# B&R Automation Studio project NAINV104C00R8L515F00 (part 34)

#### Local.var
```iecst
(*2021-05-18*)
(**)
(*Local Action, State & Status*)
VAR
	eStatus : eFBStatus := Idle;
	udiStatus : UDINT := 0;
END_VAR
(**)
(*Local Alarm*)
VAR
	tyAlmData : tyAlmDat;
	tyInfoData : tyAlmDat;
	tyInfoData1 : tyAlmDat;
	a_tyAlmText : ARRAY[10000..10099] OF tyAlmTxt := [(sAlmText:='New Recipe Not Found In Product Recipe List',sRcyText:='Create New Recipe In Product Setting.'),(sAlmText:='Product Recipe Width Not Match',sRcyText:='Check Product Width And Leader Request Width'),(sAlmText:='New Recipe Not Found In Magazine Recipe List',sRcyText:='Create New Recipe In Magazine Setting.'),(sAlmText:='New Recipe Name Empty',sRcyText:='Request Recipe Name From Leader Is Empty, Check Leader Machine'),96(0)];
END_VAR
(**)
(*Local Output*)
VAR
	bUSAllow : BOOL;
	bDSAllow : BOOL;
	bLeaderSeqCtrlInActive : BOOL;
	bProdAccDataMnl : BOOL;
	bProdUpdtDataMnl : BOOL;
	bMagAccDataMnl : BOOL;
	eTimeAct : eTimeAction;
	bWaitRlsBrd : BOOL;
	tyLeaderInfo : tyLFLeaderInfo;
	tyUpdtProdRcp : tyProdRcpParam;
END_VAR
(**)
(*Local Input*)
VAR
	udiRstErr : UDINT := 0;
	bPrep : BOOL := TRUE;
	bEn : BOOL := TRUE;
	bDis : BOOL := FALSE;
	sIPAddr : STRING[15] := '192.168.0.100';
	sMcNm : STRING[30];
	bAWPrep : BOOL := TRUE;
	bAWDis : BOOL;
	bMnlAccData : BOOL;
	bSectionLeader : BOOL;
	sMagRcpNm : STRING[30];
	diWidthLimit : DINT;
	bWidth2Prep : BOOL;
	bUSWidthChkPrep : BOOL;
	bUSWidthChkEn : BOOL;
	bUSWidthChkSen : BOOL;
	bDSWidthChkPrep : BOOL;
	bDSWidthChkEn : BOOL;
	bDSWidthChkSen : BOOL;
	bProdWidthChk : BOOL;
	bUIProdAccData : BOOL;
	bUIProdUpdtData : BOOL;
	bUIMagAccData : BOOL;
	a_tyProdRcpList : ARRAY[1..c_udiProdRcpMax] OF tyProdRcpParam;
	tyDispProdRcp : tyProdRcpParam;
	tyCurrProdRcp : tyProdRcpParam;
	sCurrMagRcpNm : STRING[30];
	eTimeStat : eTimeAction;
	eTimeStatus : eFBStatus;
	bAccNewRcpCond : BOOL;
	bUpdtNewRcpCond : BOOL;
	bAutoUpdtData : BOOL;
	sInfoMsg : STRING[200];
	bInternalUse : BOOL;
	tyInternalReqProdRcp : tyProdRcpParam;
	bNewBrdEnteredCond : BOOL;
	bOldBrdExitedCond : BOOL;
	bRlsBrd : BOOL;
	tyToLeaderProdRcp : tyProdRcpParam;
	bInternalReqProdRcpDiff : BOOL;
	bUpdtProdRcpDiff : BOOL;
	bRlsBrdProdRcpDiff : BOOL;
	sProgNm : STRING[15] := 'Follower';
	bNtSettingsLoadDone : BOOL := TRUE;
	tOnlineChkDlyTm : TIME;
	bManual : BOOL := FALSE;
	bErr : BOOL := FALSE;
	bWarning : BOOL := FALSE;
	bOps : BOOL := FALSE;
	bStandby : BOOL := FALSE;
	eAWStat : eAWAction;
END_VAR
(**)
(*Local*)
VAR
	bRstErr : BOOL;
	udiRstErrOld : UDINT;
	bInitDone : BOOL;
	bInitialDone : BOOL;
	bAutoAccData : BOOL;
	bProdRcpErr : BOOL;
	bMagRcpErr : BOOL;
	bSetTmErr : BOOL;
	bProdAccDataReq : BOOL;
	sReqProdRcpNm : STRING[254];
	diReqProdRcpWidth : DINT;
	bMagAccDataReq : BOOL;
	sReqMagRcpNm : STRING[30];
	usiProdAccDatStep : USINT;
	usiMagAccDatStep : USINT;
	usiProdUpdtDatStep : USINT;
	tyRlsBrdProdRcpNm : tyProdRcpParam;
	bNewBrdEntered : BOOL;
	bOldBrdExited : BOOL;
	i : INT;
	bSetTm : BOOL;
	fbOnlineChk : fbLFFollowerOnlineChk;
	fbFollower : fbLFFollower;
	tyLeaderToFollowerTag : tyLFLeaderToFollowerTag;
	tyFollowerToLeaderTag : tyLFFollowerToLeaderTag;
	eCurrMachineStat : eMachineStat;
	bLeaderOnline : BOOL;
	bLeaderInfo : BOOL;
	bFollowerInfo : BOOL;
	bProdRcpErrNotExist : BOOL;
	bProdRcpErrWidthMismatch : BOOL;
	bDBAOnWOAlign : BOOL;
	udiModuleNum : UDINT := 3901;
END_VAR
```

#### Act_Alarm.st
```iecst
(** 2019-04-21 **)
ACTION Act_Alarm:

	//Error
	IF EDGEPOS(eStatus = Error) THEN

		tyAlmData.sProgNm		:= p_sProgNm;
		tyAlmData.udiCode		:= udiStatus;
		tyAlmData.eSeverity		:= AlmSeverityError;
		tyAlmData.udiRunTime	:= tyAlmData.udiRunTime + 1;
		tyAlmData.bAlm			:= TRUE;
		tyAlmData.udiModuleNum  := udiModuleNum;
		g_sLFFollowerProgNm		:= p_sProgNm;
		//Get Error Message
		IF tyAlmData.udiCode < 10000 OR tyAlmData.udiCode > 10099 THEN
			tyAlmData.sAlmMsg	:= 'Unknown';
			tyAlmData.sRcyMsg	:= 'Unknown';
		ELSE
			tyAlmData.sAlmMsg	:= a_tyAlmText[tyAlmData.udiCode].sAlmText;
			tyAlmData.sRcyMsg	:= a_tyAlmText[tyAlmData.udiCode].sRcyText;
		END_IF

	ELSIF bRstErr AND (tyAlmData.udiCode <> 0) THEN

		tyAlmData.udiCode	:= 0;
		tyAlmData.eSeverity	:= AlmSeverityNA;
		tyAlmData.sAlmMsg	:= '';
		tyAlmData.sRcyMsg	:= '';
		tyAlmData.bAlm			:= FALSE;
	END_IF

END_ACTION
```

#### Act_Background.st
```iecst
(** 2021-05-18 **)
ACTION Act_Background:

	IF p_bInternalUse = TRUE THEN
		tyLeaderToFollowerTag.sReqProdRcpNm		:= p_tyInternalReqProdRcp.sRcpNm;
		IF p_bWidth2Prep THEN
			tyLeaderToFollowerTag.diReqProdRcpWidth	:= p_tyInternalReqProdRcp.diWidthInUM2;
		ELSE
			tyLeaderToFollowerTag.diReqProdRcpWidth	:= p_tyInternalReqProdRcp.diWidthInUM;
		END_IF
		tyLeaderToFollowerTag.sReqMagRcpNm		:= '';
		tyLeaderToFollowerTag.bMnlAccData		:= FALSE;
		tyLeaderToFollowerTag.bBypassMnlAccData	:= FALSE;
		tyLeaderToFollowerTag.bBlkDS			:= FALSE;
		tyLeaderToFollowerTag.bBlkUS			:= FALSE;
		tyLeaderToFollowerTag.bBypassWidthChk	:= TRUE;
		tyLeaderToFollowerTag.bSetTm			:= FALSE;
		tyLeaderToFollowerTag.dtTm				:= 0;
		tyLeaderToFollowerTag.uiTmZone			:= 0;
		tyLeaderToFollowerTag.usiRunTm			:= 0;
		tyLeaderToFollowerTag.bProdNameUSWarn	:= FALSE;
		tyLeaderToFollowerTag.bProdNameDSWarn	:= FALSE;
		tyLeaderToFollowerTag.bProdWidthUSWarn	:= FALSE;
		tyLeaderToFollowerTag.bProdWidthDSWarn	:= FALSE;
		tyLeaderToFollowerTag.bLeaderSeqCtrlInActive	:= FALSE;
	END_IF

	Act_Background_UpdtData;

	//FB
	fbFollower.tyLeaderToFollowerTag	:= tyLeaderToFollowerTag;
	fbFollower.sMcNm					:= p_sMcNm;
	fbFollower.sIPAddr					:= p_sIPAddr;
	fbFollower.bSectionLeader			:= p_bSectionLeader;
	fbFollower.sCurrProdRcpNm			:= p_tyCurrProdRcp.sRcpNm;
	fbFollower.diCurrProdWidthUS		:= p_tyCurrProdRcp.diWidthInUM;
	fbFollower.diCurrProdWidthDS		:= p_tyCurrProdRcp.diWidthInUM2;
	fbFollower.sCurrMagRcpNm			:= p_sCurrMagRcpNm;
	fbFollower.sUpdtLeaderProdRcpNm		:= p_tyToLeaderProdRcp.sRcpNm;
	fbFollower.diUpdtLeaderProdWidthUS	:= p_tyToLeaderProdRcp.diWidthInUM;
	fbFollower.diUpdtLeaderProdWidthDS	:= p_tyToLeaderProdRcp.diWidthInUM2;
	fbFollower.sUpdtLeaderMagRcpNm		:= p_sMagRcpNm;
	fbFollower.bMnlAccDat				:= p_bMnlAccData;
	fbFollower.bAWEn					:= (p_bAWPrep = TRUE) AND (p_bAWDis = FALSE);
	fbFollower.bUSWidthChkEn			:= p_bUSWidthChkPrep AND p_bUSWidthChkEn;
	fbFollower.bUSWidthChkSen			:= p_bUSWidthChkSen;
	fbFollower.bDSWidthChkEn			:= p_bDSWidthChkPrep AND p_bDSWidthChkEn;
	fbFollower.bDSWidthChkSen			:= p_bDSWidthChkSen;
	fbFollower.bProdWidthChk			:= p_bProdWidthChk;
	fbFollower.bProdRcpErr				:= bProdRcpErr;
	fbFollower.bMagRcpErr				:= bMagRcpErr;
	fbFollower.bSetTmErr				:= bSetTmErr;
	fbFollower.eCurrMachineStat			:= eCurrMachineStat;
	fbFollower.bProdChgOverActive		:= (p_eAWStat = AWActGoWidthOff);
	fbFollower.bDBAOnWOAlign			:= p_bDBAOnWOAlign;

	fbFollower(bEn := TRUE);

	tyFollowerToLeaderTag	:= fbFollower.tyFollowerToLeaderTag;
	bProdAccDataReq			:= fbFollower.bProdAccDataReq OR (p_bInternalReqProdRcpDiff = TRUE) ;
	bMagAccDataReq			:= fbFollower.bMagAccDataReq;
	bAutoAccData			:= fbFollower.bAutoAccData;

	IF p_bInternalUse THEN
		bLeaderOnline			:= TRUE;
	ELSE
		bLeaderOnline			:= tyLeaderInfo.bOnline;
	END_IF

	IF bLeaderOnline=FALSE THEN
		bUSAllow				:= TRUE;
		bDSAllow				:= TRUE;
		bLeaderSeqCtrlInActive	:= FALSE;
	ELSE
		bUSAllow				:= fbFollower.bUSAllow AND (p_bInternalReqProdRcpDiff = FALSE);
		bDSAllow				:= fbFollower.bDSAllow;
		bLeaderSeqCtrlInActive	:= tyLeaderToFollowerTag.bLeaderSeqCtrlInActive;
	END_IF

	fbOnlineChk.tyLeaderToFollowerTag	:= tyLeaderToFollowerTag;
	fbOnlineChk(bEn := TRUE);

	Act_Background_AccData;
	Act_Background_ChkRlsBrd;

	//Set Time
	IF EDGEPOS(tyLeaderToFollowerTag.bSetTm) THEN
		bSetTm	:= TRUE;
	END_IF

	IF bSetTm = TRUE THEN
		eTimeAct	:= TimeActSetTime;

		IF (p_eTimeStat = TimeActSetTime) AND (p_eTimeStatus = Done) THEN
			eTimeAct		:= TimeActIdle;
			bSetTm			:= FALSE;
		ELSIF p_eTimeStatus = Error THEN
			eTimeAct		:= TimeActIdle;
			bSetTm			:= FALSE;
		END_IF
	END_IF

	bSetTmErr	:= p_eTimeStatus = Error;

	IF (eStatus = Error) AND bRstErr THEN
		eStatus		:= Idle;
		udiStatus	:= 0;
		bProdRcpErr	:= FALSE;
		bProdRcpErrNotExist	:= FALSE;
		bProdRcpErrWidthMismatch:= FALSE;
		bMagRcpErr	:= FALSE;
	END_IF

END_ACTION
```

#### Act_Background_AccData.st
```iecst
(** 2023-02-22 **)
ACTION Act_Background_AccData:
	//Product Accept Data Request
	CASE usiProdAccDatStep OF
		0:
			//Check Error & Request Accept Data
			// If Product Name/Width Error, Check In Background To Update Data
			IF ((eStatus <> Error) AND (bProdAccDataReq = TRUE)) OR bProdRcpErr THEN
				sReqProdRcpNm		:= tyLeaderToFollowerTag.sReqProdRcpNm;
				diReqProdRcpWidth	:= tyLeaderToFollowerTag.diReqProdRcpWidth;
				usiProdAccDatStep	:= 1;
			END_IF

			IF bLeaderOnline=FALSE THEN
				tyInfoData.sProgNm		:= '';
				tyInfoData.udiCode		:= 0;
				tyInfoData.eSeverity	:= AlmSeverityNA;
				tyInfoData.sAlmMsg		:= '';

				bProdRcpErr 			:= FALSE;
				bProdRcpErrNotExist		:= FALSE;
				bProdRcpErrWidthMismatch:= FALSE;
			END_IF

		1:
			IF p_bInternalUse THEN
				usiProdAccDatStep	:= 2;
			ELSE
				//Check In List Of Recipe
				FOR i := 1 TO 2000 DO
					IF sReqProdRcpNm = '' THEN
						EXIT;
					ELSIF sReqProdRcpNm = pa_tyProdRcpList[i].sRcpNm  THEN
						EXIT;
					END_IF
				END_FOR

				IF sReqProdRcpNm = pa_tyProdRcpList[i].sRcpNm AND diReqProdRcpWidth <> pa_tyProdRcpList[i].diWidthInUM THEN
					//Width Mismatch
					bProdRcpErr := TRUE;
					bProdRcpErrWidthMismatch:= TRUE;
					bProdRcpErrNotExist		:= FALSE;
					usiProdAccDatStep	:= 0;
				ELSIF i > 2000 THEN
					//Recipe Not Exist
					bProdRcpErr := TRUE;
					bProdRcpErrNotExist	:= TRUE;
					bProdRcpErrWidthMismatch:= FALSE;
					usiProdAccDatStep	:= 0;
				ELSE
					bProdRcpErr := FALSE;
					bProdRcpErrNotExist	:= FALSE;
					bProdRcpErrWidthMismatch:= FALSE;
					usiProdAccDatStep	:= 2;
				END_IF

				//Info Message
				IF bLeaderOnline=FALSE THEN
					tyInfoData.sProgNm		:= '';
					tyInfoData.udiCode		:= 0;
					tyInfoData.eSeverity	:= AlmSeverityNA;
					tyInfoData.sAlmMsg		:= '';

					bProdRcpErr 			:= FALSE;
					bProdRcpErrNotExist		:= FALSE;
					bProdRcpErrWidthMismatch:= FALSE;
				ELSE

					IF p_bInternalUse = FALSE THEN
						IF bLeaderInfo OR bFollowerInfo THEN
							tyInfoData.sProgNm		:= p_sProgNm;
							tyInfoData.udiCode		:= 10000;
							tyInfoData.eSeverity	:= AlmSeverityInfo;
							tyInfoData.sAlmMsg		:= p_sInfoMsg;
						ELSE
							tyInfoData.sProgNm		:= '';
							tyInfoData.udiCode		:= 0;
							tyInfoData.eSeverity	:= AlmSeverityNA;
							tyInfoData.sAlmMsg		:= '';
						END_IF
					ELSE
						IF p_sInfoMsg <> '' THEN
							tyInfoData.sProgNm		:= p_sProgNm;
							tyInfoData.udiCode		:= 10000;
							tyInfoData.eSeverity	:= AlmSeverityInfo;
							tyInfoData.sAlmMsg		:= p_sInfoMsg;
						ELSE
							tyInfoData.sProgNm		:= '';
							tyInfoData.udiCode		:= 0;
							tyInfoData.eSeverity	:= AlmSeverityNA;
							tyInfoData.sAlmMsg		:= '';
						END_IF

					END_IF
				END_IF
			END_IF
		2:
			//Manual Accept Data Check
			IF bProdAccDataReq = TRUE THEN
				IF bAutoAccData = FALSE THEN
					bProdAccDataMnl	:= TRUE;

					//Info Message
					IF bLeaderOnline=FALSE THEN
						tyInfoData.sProgNm		:= '';
						tyInfoData.udiCode		:= 0;
						tyInfoData.eSeverity	:= AlmSeverityNA;
						tyInfoData.sAlmMsg		:= '';
					ELSE
						IF p_sInfoMsg <> '' THEN
							tyInfoData.sProgNm		:= p_sProgNm;
							tyInfoData.udiCode		:= 10000;
							tyInfoData.eSeverity	:= AlmSeverityInfo;
							tyInfoData.sAlmMsg		:= p_sInfoMsg;
						ELSE
							tyInfoData.sProgNm		:= '';
							tyInfoData.udiCode		:= 0;
							tyInfoData.eSeverity	:= AlmSeverityNA;
							tyInfoData.sAlmMsg		:= '';
						END_IF
					END_IF

					IF p_bUIProdAccData = TRUE THEN
						p_bUIProdAccData 	:= FALSE; //2023_07_26_Debug for Manual Accept Data automatically accept after product change many times
						bProdAccDataMnl		:= FALSE;
						usiProdAccDatStep	:= 3;
					END_IF
				ELSE
					bProdAccDataMnl		:= FALSE;
					p_bUIProdAccData	:= FALSE; //2023_07_26_Debug for Manual Accept Data automatically accept after product change many times
					usiProdAccDatStep	:= 3;
				END_IF
			ELSE
				bProdAccDataMnl		:= FALSE;
				usiProdAccDatStep	:= 6;
			END_IF

		3:
			//Accept New Recipe Condition
			IF bProdAccDataReq = TRUE THEN
				IF p_bAccNewRcpCond = TRUE THEN

					usiProdAccDatStep	:= 4;
				ELSE
					//Info Message
					IF bLeaderOnline=FALSE THEN
						tyInfoData.sProgNm		:= '';
						tyInfoData.udiCode		:= 0;
						tyInfoData.eSeverity	:= AlmSeverityNA;
						tyInfoData.sAlmMsg		:= '';
					ELSE
						IF p_sInfoMsg <> '' THEN
							tyInfoData.sProgNm		:= p_sProgNm;
							tyInfoData.udiCode		:= 10000;
							tyInfoData.eSeverity	:= AlmSeverityInfo;
							tyInfoData.sAlmMsg		:= p_sInfoMsg;
						ELSE
							tyInfoData.sProgNm		:= '';
							tyInfoData.udiCode		:= 0;
							tyInfoData.eSeverity	:= AlmSeverityNA;
							tyInfoData.sAlmMsg		:= '';
						END_IF
					END_IF
				END_IF
			ELSE
				usiProdAccDatStep	:= 6;
			END_IF

		4:
			//Accept New Recipe Name
			IF p_bInternalUse = TRUE THEN

				p_tyCurrProdRcp	:= p_tyInternalReqProdRcp;
				usiProdAccDatStep := 6;
			ELSE

				FOR i := 1 TO 2000 DO
					IF sReqProdRcpNm = '' THEN
						EXIT;
					ELSIF sReqProdRcpNm = pa_tyProdRcpList[i].sRcpNm THEN
						p_tyCurrProdRcp	:= pa_tyProdRcpList[i];

						EXIT;
					END_IF
				END_FOR

				IF i > 2000 THEN
					//Recipe Not Exist
					bProdRcpErr := TRUE;
					bProdRcpErrNotExist	:= TRUE;
				END_IF
				usiProdAccDatStep	:= 5;
			END_IF

		5:
			(* Add *)
			p_tyProdRcpCurrRcpWr 	:= p_tyCurrProdRcp;
			p_eLinkUIProdRcpAct 	:= ProdRcpActWriteCurrRcpParam;

			IF p_eProdRcpStat = ProdRcpActWriteCurrRcpParam AND p_eProdRcpStatus = Done THEN
				p_eLinkUIProdRcpAct := ProdRcpActIdle;
				usiProdAccDatStep := 6;
			END_IF

		6:
			//Clear Info Message
			tyInfoData.sProgNm		:= '';
			tyInfoData.udiCode		:= 0;
			tyInfoData.eSeverity	:= AlmSeverityNA;
			tyInfoData.sAlmMsg		:= '';

			usiProdAccDatStep	:= 0;

	END_CASE

END_ACTION
```

#### Act_Background_UpdtData.st
```iecst
(** 2019-07-04 **)
ACTION Act_Background_UpdtData:

	//Update To Leader Recipe
	CASE usiProdUpdtDatStep OF
		0:
			//Update New Recipe Condition
			IF tyUpdtProdRcp.sRcpNm <> '' THEN
				IF (p_tyCurrProdRcp.sRcpNm <> tyUpdtProdRcp.sRcpNm) OR (p_bUpdtProdRcpDiff = TRUE) THEN
					IF p_bUpdtNewRcpCond = TRUE THEN
						usiProdUpdtDatStep	:= 1;
					END_IF
				END_IF
			ELSE
				tyUpdtProdRcp	:= p_tyCurrProdRcp;
			END_IF

		1:
			//Manual Update Data Check
			IF p_bAutoUpdtData = FALSE THEN
				bProdUpdtDataMnl	:= TRUE;

				IF p_bUIProdUpdtData = TRUE THEN
					bProdUpdtDataMnl	:= FALSE;
					usiProdUpdtDatStep	:= 2;
				END_IF
			ELSE
				bProdUpdtDataMnl	:= FALSE;
				usiProdUpdtDatStep	:= 2;
			END_IF

		2:
			//Update New Recipe
			tyUpdtProdRcp	:= p_tyCurrProdRcp;

			usiProdUpdtDatStep	:= 0;

	END_CASE

END_ACTION
```

#### Act_InitGlobal.st
```iecst
(** 2020-08-06 **)
ACTION Act_InitGlobal:

	(* Always Change If Project Change *)

	//Pass Data To Link
	p_bLinkStartupRun ACCESS p_StartupRun;
	p_eLinkMcParamUSCommMod ACCESS p_McParamUSCommMod;

	p_bLinkOpsRun ACCESS p_OpsRun;
	p_bLinkConvHvBrd ACCESS p_OpsInvertHvBrd;
	p_bLinkUSWidthChkSen ACCESS p_DIUSWidthChkSen;
	p_bLinkUSWidthChkSen1 ACCESS p_DIUSWidthChkSen1;
	p_bLinkDIInvertHomeSen ACCESS p_DIInvertHomeSen;
	p_bLinkDIInvertRemoteSen ACCESS p_DIInvertRemoteSen;

	//Pass Data To Internal Use
	p_udiRstErr ACCESS p_RstErrReset;
	p_bPrep ACCESS p_NtParamLFPrep;
	p_bEn ACCESS p_McParamLFEn;
	p_sIPAddr ACCESS p_HWInfoIPAddr;
	p_sMcNm ACCESS p_McParamMcNm;
	p_bAWPrep ACCESS p_NtParamAWPrep;
	p_bAWDis ACCESS p_McParamAWDis;
	p_bMnlAccData ACCESS p_McParamMnlAccDat;
	p_bSectionLeader ACCESS p_McParamSectionLeader;
	p_diWidthLimit ACCESS p_NtParamLFWidthLimit;
	p_bUSWidthChkPrep ACCESS p_NtParamUSWidthChkPrep;
	p_bUSWidthChkEn ACCESS p_McParamUSWidthChkEn;
//	p_bUSWidthChkSen ACCESS p_DIUSWidthChkSen;
	p_bDSWidthChkPrep ACCESS p_NtParamDSWidthChkPrep;
	p_bDSWidthChkEn ACCESS p_McParamDSWidthChkEn;
	p_bDSWidthChkSen ACCESS p_DIDSWidthChkSen;
	p_bProdWidthChk ACCESS p_NtParamLFProdWidthChk;
	p_bUIProdAccData ACCESS p_UIProdAccData;
	p_bUIProdUpdtData ACCESS p_UIProdAccData;
	pa_tyProdRcpList ACCESS p_ProdRcpCurrList;
	p_tyCurrProdRcp ACCESS p_ProdRcpCurrRcp0;
	p_tyDispProdRcp ACCESS p_ProdRcpCurrRcp1;
	p_eTimeStat ACCESS p_TimeStat;
	p_eTimeStatus ACCESS p_TimeStatus;
	p_tyToLeaderProdRcp ACCESS p_Follower1UpdtProdRcp;	//Assign With Conveyor Last Zone (To Leader Completion Update)
	p_sProgNm ACCESS p_NtParamLFFollowerProgNm;
	p_bNtSettingsLoadDone ACCESS p_StartupNtSettingsLoadDone;

	p_tOnlineChkDlyTm ACCESS p_NtParamLFFllowerOnlineChkDlyTm;
	p_bManual ACCESS p_UIUIMnlMod;
	p_bErr ACCESS p_AlarmErr;
	p_bOps ACCESS p_OpsStatusRun;
	p_bStandby ACCESS p_OpsStatusStop;
	p_bWarning ACCESS p_AlarmWarning;
	p_eAWStat ACCESS p_AWOpenStat;
	p_bWidth2Prep ACCESS p_NtParamLFWidth2Prep;
	p_bDBAOnWOAlign ACCESS p_McParamDBAOnWOAlign;

	// Add for remain last Loaded product after power cycle
	p_eProdRcpStat ACCESS p_ProdRcpStat;
	p_eProdRcpStatus ACCESS p_ProdRcpStatus;
	p_eLinkUIProdRcpAct ACCESS p_UIProdRcpAct;
	p_tyProdRcpCurrRcpWr ACCESS p_UIProdRcpCurrRcpWr;

	(* Always Change If Project Change *)

END_ACTION
```

#### Act_Initial.st
```iecst
(** 2020-08-06 **)
ACTION Act_Initial:

	//Initial
	fbFollower.diWidthLimit	:= p_diWidthLimit;
	fbFollower(bEn := FALSE);

	fbOnlineChk.p_tyLeaderInfo		:= ADR(tyLeaderInfo);
	fbOnlineChk.tDlyTm				:= p_tOnlineChkDlyTm;
	fbOnlineChk(bEn := FALSE);

END_ACTION
```

#### Act_InitLocal.st
```iecst
(** 2021-05-18 **)
ACTION Act_InitLocal:

	//Input Reference Link To Local Variable
	p_udiRstErr ACCESS ADR(udiRstErr);
	p_bPrep ACCESS ADR(bPrep);
	p_bEn ACCESS ADR(bEn);
	p_bDis ACCESS ADR(bDis);
	p_sIPAddr ACCESS ADR(sIPAddr);
	p_sMcNm ACCESS ADR(sMcNm);
	p_bAWPrep ACCESS ADR(bAWPrep);
	p_bAWDis ACCESS ADR(bAWDis);
	p_bMnlAccData ACCESS ADR(bMnlAccData);
	p_bSectionLeader ACCESS ADR(bSectionLeader);
	p_sMagRcpNm ACCESS ADR(sMagRcpNm);
	p_diWidthLimit ACCESS ADR(diWidthLimit);
	p_bUSWidthChkPrep ACCESS ADR(bUSWidthChkPrep);
	p_bUSWidthChkEn ACCESS ADR(bUSWidthChkEn);
	p_bUSWidthChkSen ACCESS ADR(bUSWidthChkSen);
	p_bDSWidthChkPrep ACCESS ADR(bDSWidthChkPrep);
	p_bDSWidthChkEn ACCESS ADR(bDSWidthChkEn);
	p_bDSWidthChkSen ACCESS ADR(bDSWidthChkSen);
	p_bProdWidthChk ACCESS ADR(bProdWidthChk);
	p_bUIProdAccData ACCESS ADR(bUIProdAccData);
	p_bUIProdUpdtData ACCESS ADR(bUIProdUpdtData);
	p_bUIMagAccData ACCESS ADR(bUIMagAccData);
	pa_tyProdRcpList ACCESS ADR(a_tyProdRcpList);
	p_tyCurrProdRcp ACCESS ADR(tyCurrProdRcp);
	p_tyDispProdRcp ACCESS ADR(tyDispProdRcp);
	p_sCurrMagRcpNm ACCESS ADR(sCurrMagRcpNm);
	p_eTimeStat ACCESS ADR(eTimeStat);
	p_eTimeStatus ACCESS ADR(eTimeStatus);
	p_bAccNewRcpCond ACCESS ADR(bAccNewRcpCond);
	p_bUpdtNewRcpCond ACCESS ADR(bUpdtNewRcpCond);
	p_bAutoUpdtData ACCESS ADR(bAutoUpdtData);
	p_sInfoMsg ACCESS ADR(sInfoMsg);
	p_bInternalUse ACCESS ADR(bInternalUse);
	p_tyInternalReqProdRcp ACCESS ADR(tyInternalReqProdRcp);
	p_bNewBrdEnteredCond ACCESS ADR(bNewBrdEnteredCond);
	p_bOldBrdExitedCond ACCESS ADR(bOldBrdExitedCond);
	p_bRlsBrd ACCESS ADR(bRlsBrd);
	p_tyToLeaderProdRcp ACCESS ADR(tyToLeaderProdRcp);
	p_bInternalReqProdRcpDiff ACCESS ADR(bInternalReqProdRcpDiff);
	p_bUpdtProdRcpDiff ACCESS ADR(bUpdtProdRcpDiff);
	p_bRlsBrdProdRcpDiff ACCESS ADR(bRlsBrdProdRcpDiff);
	p_sProgNm ACCESS ADR(sProgNm);
	p_bNtSettingsLoadDone ACCESS ADR(bNtSettingsLoadDone);
	p_tOnlineChkDlyTm ACCESS ADR(tOnlineChkDlyTm);
	p_bManual ACCESS ADR(bManual);
	p_bErr ACCESS ADR(bErr);
	p_bWarning ACCESS ADR(bWarning);
	p_bOps ACCESS ADR(bOps);
	p_bStandby ACCESS ADR(bStandby);
	p_eAWStat ACCESS ADR(eAWStat);
	p_bWidth2Prep ACCESS ADR(bWidth2Prep);
	p_bDBAOnWOAlign ACCESS ADR(bDBAOnWOAlign);
END_ACTION
```

#### Act_Link.st
```iecst
(** 2021-05-18 **)
ACTION Act_Link:

	bFollowerInfo	:= tyFollowerToLeaderTag.bProdWidthErr OR bProdRcpErrNotExist OR bProdRcpErrWidthMismatch;

	bLeaderInfo		:= (tyLeaderToFollowerTag.bProdWidthUSWarn OR tyLeaderToFollowerTag.bProdWidthDSWarn
						OR ((tyLeaderToFollowerTag.bProdNameUSWarn OR tyLeaderToFollowerTag.bProdNameDSWarn)
						AND (p_bAWPrep = TRUE) AND (p_bAWDis = FALSE) AND (p_eAWStat<>AWActGoWidthOff)));

	//Info Message
	IF bFollowerInfo THEN
		IF tyFollowerToLeaderTag.bProdWidthErr = TRUE OR bProdRcpErrWidthMismatch THEN

			p_sInfoMsg		:= 'Product Recipe Width Does Not Match';
			p_sInfoMsg		:= CONCAT(p_sInfoMsg , '$r$n');
			p_sInfoMsg		:= CONCAT(p_sInfoMsg , 'Check Product Width And');
			p_sInfoMsg		:= CONCAT(p_sInfoMsg , '$r$n');
			p_sInfoMsg		:= CONCAT(p_sInfoMsg , 'Leader Request Width');

		ELSIF bProdRcpErrNotExist THEN

			p_sInfoMsg		:= 'New Product Not Found';
			p_sInfoMsg		:= CONCAT(p_sInfoMsg , '$r$n');
			p_sInfoMsg		:= CONCAT(p_sInfoMsg , 'In Product Recipe List');
			p_sInfoMsg		:= CONCAT(p_sInfoMsg , '$r$n');
			p_sInfoMsg		:= CONCAT(p_sInfoMsg , 'Create New Product');
			p_sInfoMsg		:= CONCAT(p_sInfoMsg , '$r$n');
			p_sInfoMsg		:= CONCAT(p_sInfoMsg , 'In Product Setting');
		END_IF
	ELSE

		IF (tyLeaderToFollowerTag.sReqProdRcpNm<>p_tyCurrProdRcp.sRcpNm) AND (tyLeaderToFollowerTag.sReqProdRcpNm<>'')
			AND bLeaderInfo=FALSE THEN

			p_sInfoMsg		:= 'Leader Request New Recipe';
			p_sInfoMsg		:= CONCAT(p_sInfoMsg , '$r$n');
			p_sInfoMsg		:= CONCAT(p_sInfoMsg , 'Old Recipe Name : ');
			p_sInfoMsg		:= CONCAT(p_sInfoMsg , p_tyDispProdRcp.sRcpNm);
			p_sInfoMsg		:= CONCAT(p_sInfoMsg , '$r$n');
			p_sInfoMsg		:= CONCAT(p_sInfoMsg , 'Old Recipe Width : ');
			sWidthInUMTemp	:= DINT_TO_STRING(p_tyDispProdRcp.diWidthInUM / 1000);
			p_sInfoMsg		:= CONCAT(p_sInfoMsg , sWidthInUMTemp);
			p_sInfoMsg		:= CONCAT(p_sInfoMsg , '$r$n');
			p_sInfoMsg		:= CONCAT(p_sInfoMsg , 'New Recipe Name : ');
			p_sInfoMsg		:= CONCAT(p_sInfoMsg , tyLeaderToFollowerTag.sReqProdRcpNm);
			p_sInfoMsg		:= CONCAT(p_sInfoMsg , '$r$n');
			p_sInfoMsg		:= CONCAT(p_sInfoMsg , 'New Recipe Width : ');
			sWidthInUMTemp	:= DINT_TO_STRING(tyLeaderToFollowerTag.diReqProdRcpWidth / 1000);
			p_sInfoMsg		:= CONCAT(p_sInfoMsg , sWidthInUMTemp);

		ELSIF tyLeaderToFollowerTag.bProdNameUSWarn THEN
			p_sInfoMsg		:= 'US Machine Request New Recipe';
			p_sInfoMsg		:= CONCAT(p_sInfoMsg , '$r$n');
			p_sInfoMsg		:= CONCAT(p_sInfoMsg , 'Old Recipe Name : ');
			p_sInfoMsg		:= CONCAT(p_sInfoMsg , p_tyDispProdRcp.sRcpNm);
			p_sInfoMsg		:= CONCAT(p_sInfoMsg , '$r$n');
			p_sInfoMsg		:= CONCAT(p_sInfoMsg , 'Old Recipe Width : ');
			sWidthInUMTemp	:= DINT_TO_STRING(p_tyDispProdRcp.diWidthInUM / 1000);
			p_sInfoMsg		:= CONCAT(p_sInfoMsg , sWidthInUMTemp);
			p_sInfoMsg		:= CONCAT(p_sInfoMsg , '$r$n');
			p_sInfoMsg		:= CONCAT(p_sInfoMsg , 'New Recipe Name : ');
			p_sInfoMsg		:= CONCAT(p_sInfoMsg , tyLeaderToFollowerTag.sReqProdRcpNm);
			p_sInfoMsg		:= CONCAT(p_sInfoMsg , '$r$n');
			p_sInfoMsg		:= CONCAT(p_sInfoMsg , 'New Recipe Width : ');
			sWidthInUMTemp	:= DINT_TO_STRING(tyLeaderToFollowerTag.diReqProdRcpWidth / 1000);
			p_sInfoMsg		:= CONCAT(p_sInfoMsg , sWidthInUMTemp);

		ELSIF tyLeaderToFollowerTag.bProdNameDSWarn THEN
			p_sInfoMsg		:= 'Different Recipe';
			p_sInfoMsg		:= CONCAT(p_sInfoMsg , '$r$n');
			p_sInfoMsg		:= CONCAT(p_sInfoMsg , 'From DS Machine');
			p_sInfoMsg		:= CONCAT(p_sInfoMsg , '$r$n');
			p_sInfoMsg		:= CONCAT(p_sInfoMsg , 'Current Recipe Name : ');
			p_sInfoMsg		:= CONCAT(p_sInfoMsg , p_tyCurrProdRcp.sRcpNm);
			p_sInfoMsg		:= CONCAT(p_sInfoMsg , '$r$n');
			p_sInfoMsg		:= CONCAT(p_sInfoMsg , 'Current Recipe Width : ');
			sWidthInUMTemp	:= DINT_TO_STRING(p_tyCurrProdRcp.diWidthInUM2 / 1000);
			p_sInfoMsg		:= CONCAT(p_sInfoMsg , sWidthInUMTemp);

		ELSIF tyLeaderToFollowerTag.bProdWidthUSWarn THEN
			p_sInfoMsg		:= 'Product Recipe Width Does Not Match';
			p_sInfoMsg		:= CONCAT(p_sInfoMsg , '$r$n');
			p_sInfoMsg		:= CONCAT(p_sInfoMsg , 'Check Product Width And');
			p_sInfoMsg		:= CONCAT(p_sInfoMsg , '$r$n');
			p_sInfoMsg		:= CONCAT(p_sInfoMsg , 'Leader Request Width');

		ELSIF tyLeaderToFollowerTag.bProdWidthDSWarn THEN
			p_sInfoMsg		:= 'Same Recipe : ';
			p_sInfoMsg		:= CONCAT(p_sInfoMsg , p_tyDispProdRcp.sRcpNm);
			p_sInfoMsg		:= CONCAT(p_sInfoMsg , '$r$n');
			p_sInfoMsg		:= CONCAT(p_sInfoMsg , 'But Different Width');
			p_sInfoMsg		:= CONCAT(p_sInfoMsg , '$r$n');
			p_sInfoMsg		:= CONCAT(p_sInfoMsg , 'With DS Machine');
			p_sInfoMsg		:= CONCAT(p_sInfoMsg , '$r$n');
			p_sInfoMsg		:= CONCAT(p_sInfoMsg , 'Machine Outgoing Width : ');
			sWidthInUMTemp	:= DINT_TO_STRING(p_tyDispProdRcp.diWidthInUM2 / 1000);
			p_sInfoMsg		:= CONCAT(p_sInfoMsg , sWidthInUMTemp);

		END_IF
	END_IF

	//Accept New Recipe Condition (Before Loaded New Recipe)
	p_bAccNewRcpCond	:= p_bLinkOpsRun = TRUE AND p_bLinkConvHvBrd = FALSE;

	//Update New Recipe Condition (After Loaded New Recipe)
	p_bUpdtNewRcpCond	:= TRUE;

	//Recipe Different
	//p_bInternalReqProdRcpDiff	:= memcmp(ADR(p_tyCurrProdRcp) , ADR(p_tyInternalReqProdRcp) , SIZEOF(p_tyCurrProdRcp)) <> 0;
	//p_bUpdtProdRcpDiff		:= memcmp(ADR(p_tyCurrProdRcp) , ADR(tyUpdtProdRcp) , SIZEOF(p_tyCurrProdRcp)) <> 0;
	//p_bRlsBrdProdRcpDiff		:= memcmp(ADR(p_tyCurrProdRcp) , ADR(tyRlsBrdProdRcpNm) , SIZEOF(p_tyCurrProdRcp)) <> 0;

	IF p_bErr THEN
		eCurrMachineStat := InError;
	ELSE
		IF p_bWarning THEN
			eCurrMachineStat := Warning;
		ELSE
			IF p_bOps THEN
				eCurrMachineStat := Run;
			ELSE
				IF p_bManual THEN
					eCurrMachineStat := Manual;
				ELSE
					eCurrMachineStat := Stop;
				END_IF
			END_IF
		END_IF
	END_IF

	//US width check sensor selection
	IF p_bLinkDIInvertHomeSen THEN
		p_bUSWidthChkSen := p_bLinkUSWidthChkSen;
	ELSIF p_bLinkDIInvertRemoteSen THEN
		p_bUSWidthChkSen := p_bLinkUSWidthChkSen1;
	END_IF

END_ACTION
```

#### Act_LinkEn.st
```iecst
(** 2019-04-26 **)
ACTION Act_LinkEn:

	//Link bPrep, bEn & bDis
	p_bDis	:= (p_bLinkStartupRun = TRUE) OR (p_eLinkMcParamUSCommMod = McSetCommModHermes);

END_ACTION
```

#### Act_Main_Disable.st
```iecst
(** 2021-05-18 **)
ACTION Act_Main_Disable:

	bUSAllow			:= TRUE;
	bDSAllow			:= TRUE;
	bProdAccDataMnl		:= FALSE;
	bProdUpdtDataMnl	:= FALSE;
	bMagAccDataMnl		:= FALSE;
	bWaitRlsBrd			:= FALSE;

	usiProdAccDatStep		:= 0;
	usiProdUpdtDatStep		:= 0;
	tyInfoData.sProgNm		:= '';
	tyInfoData.udiCode		:= 0;
	tyInfoData.eSeverity	:= AlmSeverityNA;
	tyInfoData.sAlmMsg		:= '';

	usiMagAccDatStep		:= 0;
	tyInfoData1.sProgNm		:= '';
	tyInfoData1.udiCode		:= 0;
	tyInfoData1.eSeverity	:= AlmSeverityNA;
	tyInfoData1.sAlmMsg		:= '';

	bSetTm		:= FALSE;

	eStatus		:= Idle;
	udiStatus	:= 0;
	bProdRcpErr	:= FALSE;
	bMagRcpErr	:= FALSE;
	bLeaderSeqCtrlInActive	:= FALSE;

	bProdRcpErrNotExist		:= FALSE;
	bProdRcpErrWidthMismatch:= FALSE;

END_ACTION
```

#### Cyclic.st
```iecst
(** 2019-04-21 **)
PROGRAM _CYCLIC

	IF bInitDone = FALSE THEN
		bInitDone	:= TRUE;

		Act_InitLocal;
		Act_InitGlobal;

	ELSIF bInitialDone = FALSE THEN
		IF p_bNtSettingsLoadDone = TRUE THEN
			bInitialDone	:= TRUE;

			Act_Initial;
		END_IF

	ELSE

		Act_RstErr;
		Act_LinkEn;

		IF (p_bPrep = TRUE) AND (p_bEn = TRUE) AND (p_bDis = FALSE) THEN
			Act_Link;
			Act_Background;

		ELSE
			Act_Main_Disable;

		END_IF

		Act_Alarm;

	END_IF

END_PROGRAM
```

#### Init.st
```iecst
(** 2020-08-06 **)
PROGRAM _INIT

	(* Always Change If Project Change *)

	//Physical Configuration
	bAutoUpdtData	:= TRUE;
	bInternalUse	:= FALSE;

	//Pass Address To Global Address For External Use
	//Action, State & Status
	p_LFFollowerStatus	:= ADR(eStatus);

	//Alarm
	p_LFFollowerAlmData		:= ADR(tyAlmData);
	p_LFFollowerInfoData	:= ADR(tyInfoData);
	p_LFFollowerInfoData1	:= ADR(tyInfoData1);

	//Output
	p_LFFollowerUSAllow			:= ADR(bUSAllow);
	p_LFFollowerDSAllow			:= ADR(bDSAllow);
	p_LFFollowerProdAccDataMnl	:= ADR(bProdAccDataMnl);
	p_LFFollowerProdUpdtDataMnl	:= ADR(bProdUpdtDataMnl);
	p_LFFollowerMagAccDataMnl	:= ADR(bMagAccDataMnl);
	p_LFFollowerTimeAct			:= ADR(eTimeAct);
	p_LFFollowerSetDT			:= ADR(tyLeaderToFollowerTag.dtTm);
	p_LFFollowerWaitRlsBrd		:= ADR(bWaitRlsBrd);
	p_LFFollowerUpdtProdRcp		:= ADR(tyUpdtProdRcp);
	p_LFFollowerLdrSeqCtrlInActive	:= ADR(bLeaderSeqCtrlInActive);

	(* Always Change If Project Change *)

END_PROGRAM
```

### Follower1.var - Change By Project
```iecst
(*2019-06-27*)
(**)
(*Action & State & Status*)
VAR
	p_Follower1Status : UDINT;
END_VAR
(**)
(*Alarm*)
VAR
	p_Follower1AlmData : UDINT;
	p_Follower1InfoData : UDINT;
	p_Follower1InfoData1 : UDINT;
END_VAR
(**)
(*Output*)
VAR
	p_Follower1USAllow : UDINT;
	p_Follower1DSAllow : UDINT;
	p_Follower1ProdAccDataMnl : UDINT;
	p_Follower1ProdUpdtDataMnl : UDINT;
	p_Follower1MagAccDataMnl : UDINT;
	p_Follower1TimeAct : UDINT;
	p_Follower1SetDT : UDINT;
	p_Follower1WaitRlsBrd : UDINT;
	p_Follower1UpdtProdRcp : UDINT;
END_VAR
```

### Program Logical/LF/Follower1 (IEC, version 1.00.0) - 1.00.0 - NtHermes v5.00.0 , NtTCP v5.00.0 , NtMessage v5.00.0

#### Init.st - Change By Project
```iecst
(** 2019-06-27 **)
PROGRAM _INIT

	(* Always Change If Project Change *)

	//Physical Configuration
	bAutoUpdtData	:= TRUE;
	bInternalUse	:= TRUE;

	//Pass Address To Global Address For External Use
	//Action, State & Status
	p_Follower1Status	:= ADR(eStatus);

	//Alarm
	p_Follower1AlmData			:= ADR(tyAlmData);
	p_Follower1InfoData			:= ADR(tyInfoData);
	p_Follower1InfoData1		:= ADR(tyInfoData1);

	//Output
	p_Follower1USAllow			:= ADR(bUSAllow);
	p_Follower1DSAllow			:= ADR(bDSAllow);
	p_Follower1ProdAccDataMnl	:= ADR(bProdAccDataMnl);
	p_Follower1ProdUpdtDataMnl	:= ADR(bProdUpdtDataMnl);
	p_Follower1MagAccDataMnl	:= ADR(bMagAccDataMnl);
	p_Follower1TimeAct			:= ADR(eTimeAct);
	p_Follower1SetDT			:= ADR(tyLeaderToFollowerTag.dtTm);
	p_Follower1WaitRlsBrd		:= ADR(bWaitRlsBrd);
	p_Follower1UpdtProdRcp		:= ADR(tyUpdtProdRcp);

	(* Always Change If Project Change *)

END_PROGRAM
```

#### Act_InitGlobal.st - Change By Project
```iecst
(** 2020-08-06 **)
ACTION Act_InitGlobal:

	(* Always Change If Project Change *)

	//Pass Data To Link
	p_bLinkStartupRun ACCESS p_StartupRun;

	p_bLinkOpsRun ACCESS p_OpsRun;
	p_bLinkOpsInvertStepInitDone ACCESS p_OpsInvertStepInitDone;
	p_bLinkConvHvBrd ACCESS p_OpsInvertHvBrd;
	p_eLinkOpsInvertCurrPos ACCESS p_OpsInvertInvertCurrPos;
	p_bLinkUSWidthChkSen ACCESS p_DIUSWidthChkSen;
	p_bLinkUSWidthChkSen1 ACCESS p_DIUSWidthChkSen1;
	p_bLinkDIInvertHomeSen ACCESS p_DIInvertHomeSen;
	p_bLinkDIInvertRemoteSen ACCESS p_DIInvertRemoteSen;

	//Pass Data To Internal Use
	p_udiRstErr ACCESS p_RstErrReset;
	p_sIPAddr ACCESS p_HWInfoIPAddr;
	p_sMcNm ACCESS p_McParamMcNm;
	p_bUSWidthChkPrep ACCESS p_NtParamUSWidthChkPrep;
	p_bUSWidthChkEn ACCESS p_McParamUSWidthChkEn;
//	p_bUSWidthChkSen ACCESS p_DIUSWidthChkSen;
	p_bDSWidthChkPrep ACCESS p_NtParamDSWidthChkPrep;
	p_bDSWidthChkEn ACCESS p_McParamDSWidthChkEn;
	p_bDSWidthChkSen ACCESS p_DIDSWidthChkSen;
	p_tyCurrProdRcp ACCESS p_ProdRcpCurrRcp1;
	p_tyInternalReqProdRcp ACCESS p_ProdRcpCurrRcp0; //Follower 1 Assign With Default Recipe
	p_bRlsBrd ACCESS p_UIRlsNewProd;
	p_sProgNm ACCESS p_NtParamFollower1ProgNm;
	p_bNtSettingsLoadDone ACCESS p_StartupNtSettingsLoadDone;

	p_bWidth2Prep ACCESS p_NtParamLFWidth2Prep;

	// Add for remain last Loaded product after power cycle
	p_eProdRcpStat ACCESS p_ProdRcpStat;
	p_eProdRcpStatus ACCESS p_ProdRcpStatus;
	p_eLinkUIProdRcpAct ACCESS p_UIProdRcpAct;
	p_tyProdRcpCurrRcpWr ACCESS p_UIProdRcpCurrRcpWr;

	(* Always Change If Project Change *)
END_ACTION
```

#### InputRef_Link.var - Change By Project
```iecst
(*2019-05-07*)
(**)
VAR
	p_bLinkStartupRun : REFERENCE TO BOOL;
END_VAR
(**)
VAR
	p_bLinkOpsRun : REFERENCE TO BOOL;
	p_bLinkOpsInvertStepInitDone : REFERENCE TO BOOL;
	p_eLinkOpsInvertCurrPos : REFERENCE TO eInvertPos;
	p_bLinkConvHvBrd : REFERENCE TO BOOL;
	p_bLinkUSWidthChkSen : REFERENCE TO BOOL;
	p_bLinkUSWidthChkSen1 : REFERENCE TO BOOL;
	p_bLinkDIInvertHomeSen : REFERENCE TO BOOL;
	p_bLinkDIInvertRemoteSen : REFERENCE TO BOOL;
END_VAR
(**)
VAR
	p_eProdRcpStatus : REFERENCE TO eFBStatus;
	p_eLinkUIProdRcpAct : REFERENCE TO eProdRcpAction;
	p_eProdRcpStat : REFERENCE TO eProdRcpAction;
	p_tyProdRcpCurrRcpWr : REFERENCE TO tyProdRcpParam;
END_VAR
```

#### Act_LinkEn.st - Change By Project
```iecst
(** 2019-04-26 **)
ACTION Act_LinkEn:

	//Link bPrep, bEn & bDis
	//p_bDis	:= (p_bLinkStartupRun = TRUE);

END_ACTION
```

#### Act_Link.st - Change By Project
```iecst
(** 2019-07-04 **)
ACTION Act_Link:

	//Temporary (Recipe No Save)
	IF p_tyCurrProdRcp.sRcpNm = '' AND p_tyCurrProdRcp.diWidthInUM = 0 THEN
		p_tyCurrProdRcp	:= p_tyInternalReqProdRcp;
	END_IF

	//Info Message
	p_sInfoMsg	:= '';

	//Accept New Recipe Condition (Before Loaded New Recipe)
	p_bAccNewRcpCond	:= (p_bLinkOpsRun = TRUE) AND (p_bLinkOpsInvertStepInitDone = TRUE) AND (p_bLinkConvHvBrd = FALSE) AND (p_eLinkOpsInvertCurrPos<>InvertPosInvalid);

	//Update New Recipe Condition (After Loaded New Recipe)
	p_bUpdtNewRcpCond	:= TRUE;

	//Recipe Different
	p_bInternalReqProdRcpDiff	:= memcmp(ADR(p_tyCurrProdRcp) , ADR(p_tyInternalReqProdRcp) , SIZEOF(p_tyCurrProdRcp)) <> 0;
	p_bUpdtProdRcpDiff			:= memcmp(ADR(p_tyCurrProdRcp) , ADR(tyUpdtProdRcp) , SIZEOF(p_tyCurrProdRcp)) <> 0;
	p_bRlsBrdProdRcpDiff		:= memcmp(ADR(p_tyCurrProdRcp) , ADR(tyRlsBrdProdRcpNm) , SIZEOF(p_tyCurrProdRcp)) <> 0;

	//Release New Product Condition
	p_bNewBrdEnteredCond	:= (p_bLinkOpsInvertStepInitDone = TRUE) AND (p_bLinkConvHvBrd = TRUE);
	p_bOldBrdExitedCond		:= (p_bLinkOpsInvertStepInitDone = TRUE) AND (p_bLinkConvHvBrd = FALSE);

	//US width check sensor selection
	IF p_bLinkDIInvertHomeSen THEN
		p_bUSWidthChkSen := p_bLinkUSWidthChkSen;
	ELSIF p_bLinkDIInvertRemoteSen THEN
		p_bUSWidthChkSen := p_bLinkUSWidthChkSen1;
	END_IF

END_ACTION
```

#### Act_RstErr.st - Do Not Change!!!
```iecst
(** 2019-04-21 **)
ACTION Act_RstErr:

	IF p_udiRstErr <> udiRstErrOld THEN
		bRstErr			:= TRUE;
		udiRstErrOld	:= p_udiRstErr;
	ELSE
		bRstErr			:= FALSE;
	END_IF

END_ACTION
```

#### Act_InitLocal.st - Do Not Change!!!
```iecst
(** 2020-08-06 **)
ACTION Act_InitLocal:

	//Input Reference Link To Local Variable
	p_udiRstErr ACCESS ADR(udiRstErr);
	p_bPrep ACCESS ADR(bPrep);
	p_bEn ACCESS ADR(bEn);
	p_bDis ACCESS ADR(bDis);
	p_sIPAddr ACCESS ADR(sIPAddr);
	p_sMcNm ACCESS ADR(sMcNm);
	p_bAWPrep ACCESS ADR(bAWPrep);
	p_bAWDis ACCESS ADR(bAWDis);
	p_bMnlAccData ACCESS ADR(bMnlAccData);
	p_bSectionLeader ACCESS ADR(bSectionLeader);
	p_sMagRcpNm ACCESS ADR(sMagRcpNm);
	p_diWidthLimit ACCESS ADR(diWidthLimit);
	p_bUSWidthChkPrep ACCESS ADR(bUSWidthChkPrep);
	p_bUSWidthChkEn ACCESS ADR(bUSWidthChkEn);
	p_bUSWidthChkSen ACCESS ADR(bUSWidthChkSen);
	p_bDSWidthChkPrep ACCESS ADR(bDSWidthChkPrep);
	p_bDSWidthChkEn ACCESS ADR(bDSWidthChkEn);
	p_bDSWidthChkSen ACCESS ADR(bDSWidthChkSen);
	p_bProdWidthChk ACCESS ADR(bProdWidthChk);
	p_bUIProdAccData ACCESS ADR(bUIProdAccData);
	p_bUIProdUpdtData ACCESS ADR(bUIProdUpdtData);
	p_bUIMagAccData ACCESS ADR(bUIMagAccData);
	pa_tyProdRcpList ACCESS ADR(a_tyProdRcpList);
	p_tyCurrProdRcp ACCESS ADR(tyCurrProdRcp);
	p_sCurrMagRcpNm ACCESS ADR(sCurrMagRcpNm);
	p_eTimeStat ACCESS ADR(eTimeStat);
	p_eTimeStatus ACCESS ADR(eTimeStatus);
	p_bAccNewRcpCond ACCESS ADR(bAccNewRcpCond);
	p_bUpdtNewRcpCond ACCESS ADR(bUpdtNewRcpCond);
	p_bAutoUpdtData ACCESS ADR(bAutoUpdtData);
	p_sInfoMsg ACCESS ADR(sInfoMsg);
	p_bInternalUse ACCESS ADR(bInternalUse);
	p_tyInternalReqProdRcp ACCESS ADR(tyInternalReqProdRcp);
	p_bNewBrdEnteredCond ACCESS ADR(bNewBrdEnteredCond);
	p_bOldBrdExitedCond ACCESS ADR(bOldBrdExitedCond);
	p_bRlsBrd ACCESS ADR(bRlsBrd);
	p_tyToLeaderProdRcp ACCESS ADR(tyToLeaderProdRcp);
	p_bInternalReqProdRcpDiff ACCESS ADR(bInternalReqProdRcpDiff);
	p_bUpdtProdRcpDiff ACCESS ADR(bUpdtProdRcpDiff);
	p_bRlsBrdProdRcpDiff ACCESS ADR(bRlsBrdProdRcpDiff);
	p_sProgNm ACCESS ADR(sProgNm);
	p_bNtSettingsLoadDone ACCESS ADR(bNtSettingsLoadDone);
	p_tOnlineChkDlyTm ACCESS ADR(tOnlineChkDlyTm);
	p_bManual ACCESS ADR(bManual);
	p_bErr ACCESS ADR(bErr);
	p_bWarning ACCESS ADR(bWarning);
	p_bOps ACCESS ADR(bOps);
	p_bStandby ACCESS ADR(bStandby);
	p_eAWStat ACCESS ADR(eAWStat);
	p_bWidth2Prep ACCESS ADR(bWidth2Prep);
	p_bDBAOnWOAlign ACCESS ADR(bDBAOnWOAlign);
END_ACTION
```

#### Act_Background.st - Do Not Change!!!
```iecst
(** 2021-05-18 **)
ACTION Act_Background:

	IF p_bInternalUse = TRUE THEN
		tyLeaderToFollowerTag.sReqProdRcpNm		:= p_tyInternalReqProdRcp.sRcpNm;
		IF p_bWidth2Prep THEN
			tyLeaderToFollowerTag.diReqProdRcpWidth	:= p_tyInternalReqProdRcp.diWidthInUM2;
		ELSE
			tyLeaderToFollowerTag.diReqProdRcpWidth	:= p_tyInternalReqProdRcp.diWidthInUM;
		END_IF
		tyLeaderToFollowerTag.sReqMagRcpNm		:= '';
		tyLeaderToFollowerTag.bMnlAccData		:= FALSE;
		tyLeaderToFollowerTag.bBypassMnlAccData	:= FALSE;
		tyLeaderToFollowerTag.bBlkDS			:= FALSE;
		tyLeaderToFollowerTag.bBlkUS			:= FALSE;
		tyLeaderToFollowerTag.bBypassWidthChk	:= TRUE;
		tyLeaderToFollowerTag.bSetTm			:= FALSE;
		tyLeaderToFollowerTag.dtTm				:= 0;
		tyLeaderToFollowerTag.uiTmZone			:= 0;
		tyLeaderToFollowerTag.usiRunTm			:= 0;
		tyLeaderToFollowerTag.bProdNameUSWarn	:= FALSE;
		tyLeaderToFollowerTag.bProdNameDSWarn	:= FALSE;
		tyLeaderToFollowerTag.bProdWidthUSWarn	:= FALSE;
		tyLeaderToFollowerTag.bProdWidthDSWarn	:= FALSE;
		tyLeaderToFollowerTag.bLeaderSeqCtrlInActive	:= FALSE;
	END_IF

	Act_Background_UpdtData;

	//FB
	fbFollower.tyLeaderToFollowerTag	:= tyLeaderToFollowerTag;
	fbFollower.sMcNm					:= p_sMcNm;
	fbFollower.sIPAddr					:= p_sIPAddr;
	fbFollower.bSectionLeader			:= p_bSectionLeader;
	fbFollower.sCurrProdRcpNm			:= p_tyCurrProdRcp.sRcpNm;
	fbFollower.diCurrProdWidthUS		:= p_tyCurrProdRcp.diWidthInUM;
	fbFollower.diCurrProdWidthDS		:= p_tyCurrProdRcp.diWidthInUM2;
	fbFollower.sCurrMagRcpNm			:= p_sCurrMagRcpNm;
	fbFollower.sUpdtLeaderProdRcpNm		:= p_tyToLeaderProdRcp.sRcpNm;
	fbFollower.diUpdtLeaderProdWidthUS	:= p_tyToLeaderProdRcp.diWidthInUM;
	fbFollower.diUpdtLeaderProdWidthDS	:= p_tyToLeaderProdRcp.diWidthInUM2;
	fbFollower.sUpdtLeaderMagRcpNm		:= p_sMagRcpNm;
	fbFollower.bMnlAccDat				:= p_bMnlAccData;
	fbFollower.bAWEn					:= (p_bAWPrep = TRUE) AND (p_bAWDis = FALSE);
	fbFollower.bUSWidthChkEn			:= p_bUSWidthChkPrep AND p_bUSWidthChkEn;
	fbFollower.bUSWidthChkSen			:= p_bUSWidthChkSen;
	fbFollower.bDSWidthChkEn			:= p_bDSWidthChkPrep AND p_bDSWidthChkEn;
	fbFollower.bDSWidthChkSen			:= p_bDSWidthChkSen;
	fbFollower.bProdWidthChk			:= p_bProdWidthChk;
	fbFollower.bProdRcpErr				:= bProdRcpErr;
	fbFollower.bMagRcpErr				:= bMagRcpErr;
	fbFollower.bSetTmErr				:= bSetTmErr;
	fbFollower.eCurrMachineStat			:= eCurrMachineStat;
	fbFollower.bProdChgOverActive		:= (p_eAWStat = AWActGoWidthOff);
	fbFollower.bDBAOnWOAlign			:= p_bDBAOnWOAlign;

	fbFollower(bEn := TRUE);

	tyFollowerToLeaderTag	:= fbFollower.tyFollowerToLeaderTag;
	bProdAccDataReq			:= fbFollower.bProdAccDataReq OR (p_bInternalReqProdRcpDiff = TRUE) ;
	bMagAccDataReq			:= fbFollower.bMagAccDataReq;
	bAutoAccData			:= fbFollower.bAutoAccData;

	IF p_bInternalUse THEN
		bLeaderOnline			:= TRUE;
	ELSE
		bLeaderOnline			:= tyLeaderInfo.bOnline;
	END_IF

	IF bLeaderOnline=FALSE THEN
		bUSAllow				:= TRUE;
		bDSAllow				:= TRUE;
		bLeaderSeqCtrlInActive	:= FALSE;
	ELSE
		bUSAllow				:= fbFollower.bUSAllow AND (p_bInternalReqProdRcpDiff = FALSE);
		bDSAllow				:= fbFollower.bDSAllow;
		bLeaderSeqCtrlInActive	:= tyLeaderToFollowerTag.bLeaderSeqCtrlInActive;
	END_IF

	fbOnlineChk.tyLeaderToFollowerTag	:= tyLeaderToFollowerTag;
	fbOnlineChk(bEn := TRUE);

	Act_Background_AccData;
	Act_Background_ChkRlsBrd;

	//Set Time
	IF EDGEPOS(tyLeaderToFollowerTag.bSetTm) THEN
		bSetTm	:= TRUE;
	END_IF

	IF bSetTm = TRUE THEN
		eTimeAct	:= TimeActSetTime;

		IF (p_eTimeStat = TimeActSetTime) AND (p_eTimeStatus = Done) THEN
			eTimeAct		:= TimeActIdle;
			bSetTm			:= FALSE;
		ELSIF p_eTimeStatus = Error THEN
			eTimeAct		:= TimeActIdle;
			bSetTm			:= FALSE;
		END_IF
	END_IF

	bSetTmErr	:= p_eTimeStatus = Error;

	IF (eStatus = Error) AND bRstErr THEN
		eStatus		:= Idle;
		udiStatus	:= 0;
		bProdRcpErr	:= FALSE;
		bProdRcpErrNotExist	:= FALSE;
		bProdRcpErrWidthMismatch:= FALSE;
		bMagRcpErr	:= FALSE;
	END_IF

END_ACTION
```

#### Act_Background_ChkRlsBrd.st - Do Not Change!!!
```iecst
(** 2019-07-04 **)
ACTION Act_Background_ChkRlsBrd:

	IF tyRlsBrdProdRcpNm.sRcpNm = '' THEN
		tyRlsBrdProdRcpNm	:= p_tyCurrProdRcp;

	ELSIF (tyRlsBrdProdRcpNm.sRcpNm <> p_tyCurrProdRcp.sRcpNm) OR (p_bRlsBrdProdRcpDiff = TRUE) THEN

		IF p_bNewBrdEnteredCond = TRUE THEN
			bNewBrdEntered	:= TRUE;
		END_IF

		IF p_bOldBrdExitedCond = TRUE THEN
			bOldBrdExited	:= TRUE;
		END_IF

		IF bNewBrdEntered AND bOldBrdExited THEN
			bWaitRlsBrd	:= TRUE;
		END_IF

		IF bWaitRlsBrd AND p_bRlsBrd THEN
			tyRlsBrdProdRcpNm	:= p_tyCurrProdRcp;
		END_IF

	ELSE
		bNewBrdEntered	:= FALSE;
		bOldBrdExited	:= FALSE;
		bWaitRlsBrd		:= FALSE;

	END_IF

END_ACTION
```

#### Act_Background_AccData.st - Do Not Change!!!
```iecst
(** 2023-02-22 **)
ACTION Act_Background_AccData:
	//Product Accept Data Request
	CASE usiProdAccDatStep OF
		0:
			//Check Error & Request Accept Data
			// If Product Name/Width Error, Check In Background To Update Data
			IF ((eStatus <> Error) AND (bProdAccDataReq = TRUE)) OR bProdRcpErr THEN
				sReqProdRcpNm		:= tyLeaderToFollowerTag.sReqProdRcpNm;
				diReqProdRcpWidth	:= tyLeaderToFollowerTag.diReqProdRcpWidth;
				usiProdAccDatStep	:= 1;
			END_IF

			IF bLeaderOnline=FALSE THEN
				tyInfoData.sProgNm		:= '';
				tyInfoData.udiCode		:= 0;
				tyInfoData.eSeverity	:= AlmSeverityNA;
				tyInfoData.sAlmMsg		:= '';

				bProdRcpErr 			:= FALSE;
				bProdRcpErrNotExist		:= FALSE;
				bProdRcpErrWidthMismatch:= FALSE;
			END_IF

		1:
			IF p_bInternalUse THEN
				usiProdAccDatStep	:= 2;
			ELSE
				//Check In List Of Recipe
				FOR i := 1 TO 2000 DO
					IF sReqProdRcpNm = '' THEN
						EXIT;
					ELSIF sReqProdRcpNm = pa_tyProdRcpList[i].sRcpNm  THEN
						EXIT;
					END_IF
				END_FOR

				IF sReqProdRcpNm = pa_tyProdRcpList[i].sRcpNm AND diReqProdRcpWidth <> pa_tyProdRcpList[i].diWidthInUM THEN
					//Width Mismatch
					bProdRcpErr := TRUE;
					bProdRcpErrWidthMismatch:= TRUE;
					bProdRcpErrNotExist		:= FALSE;
					usiProdAccDatStep	:= 0;
				ELSIF i > 2000 THEN
					//Recipe Not Exist
					bProdRcpErr := TRUE;
					bProdRcpErrNotExist	:= TRUE;
					bProdRcpErrWidthMismatch:= FALSE;
					usiProdAccDatStep	:= 0;
				ELSE
					bProdRcpErr := FALSE;
					bProdRcpErrNotExist	:= FALSE;
					bProdRcpErrWidthMismatch:= FALSE;
					usiProdAccDatStep	:= 2;
				END_IF

				//Info Message
				IF bLeaderOnline=FALSE THEN
					tyInfoData.sProgNm		:= '';
					tyInfoData.udiCode		:= 0;
					tyInfoData.eSeverity	:= AlmSeverityNA;
					tyInfoData.sAlmMsg		:= '';

					bProdRcpErr 			:= FALSE;
					bProdRcpErrNotExist		:= FALSE;
					bProdRcpErrWidthMismatch:= FALSE;
				ELSE

					IF p_bInternalUse = FALSE THEN
						IF bLeaderInfo OR bFollowerInfo THEN
							tyInfoData.sProgNm		:= p_sProgNm;
							tyInfoData.udiCode		:= 10000;
							tyInfoData.eSeverity	:= AlmSeverityInfo;
							tyInfoData.sAlmMsg		:= p_sInfoMsg;
						ELSE
							tyInfoData.sProgNm		:= '';
							tyInfoData.udiCode		:= 0;
							tyInfoData.eSeverity	:= AlmSeverityNA;
							tyInfoData.sAlmMsg		:= '';
						END_IF
					ELSE
						IF p_sInfoMsg <> '' THEN
							tyInfoData.sProgNm		:= p_sProgNm;
							tyInfoData.udiCode		:= 10000;
							tyInfoData.eSeverity	:= AlmSeverityInfo;
							tyInfoData.sAlmMsg		:= p_sInfoMsg;
						ELSE
							tyInfoData.sProgNm		:= '';
							tyInfoData.udiCode		:= 0;
							tyInfoData.eSeverity	:= AlmSeverityNA;
							tyInfoData.sAlmMsg		:= '';
						END_IF

					END_IF
				END_IF
			END_IF
		2:
			//Manual Accept Data Check
			IF bProdAccDataReq = TRUE THEN
				IF bAutoAccData = FALSE THEN
					bProdAccDataMnl	:= TRUE;

					//Info Message
					IF bLeaderOnline=FALSE THEN
						tyInfoData.sProgNm		:= '';
						tyInfoData.udiCode		:= 0;
						tyInfoData.eSeverity	:= AlmSeverityNA;
						tyInfoData.sAlmMsg		:= '';
					ELSE
						IF p_sInfoMsg <> '' THEN
							tyInfoData.sProgNm		:= p_sProgNm;
							tyInfoData.udiCode		:= 10000;
							tyInfoData.eSeverity	:= AlmSeverityInfo;
							tyInfoData.sAlmMsg		:= p_sInfoMsg;
						ELSE
							tyInfoData.sProgNm		:= '';
							tyInfoData.udiCode		:= 0;
							tyInfoData.eSeverity	:= AlmSeverityNA;
							tyInfoData.sAlmMsg		:= '';
						END_IF
					END_IF

					IF p_bUIProdAccData = TRUE THEN
						p_bUIProdAccData 	:= FALSE; //2023_07_26_Debug for Manual Accept Data automatically accept after product change many times
						bProdAccDataMnl		:= FALSE;
						usiProdAccDatStep	:= 3;
					END_IF
				ELSE
					bProdAccDataMnl		:= FALSE;
					p_bUIProdAccData 	:= FALSE; //2023_07_26_Debug for Manual Accept Data automatically accept after product change many times
					usiProdAccDatStep	:= 3;
				END_IF
			ELSE
				bProdAccDataMnl		:= FALSE;
				usiProdAccDatStep	:= 6;
			END_IF

		3:
			//Accept New Recipe Condition
			IF bProdAccDataReq = TRUE THEN
				IF p_bAccNewRcpCond = TRUE THEN

					usiProdAccDatStep	:= 4;
				ELSE
					//Info Message
					IF bLeaderOnline=FALSE THEN
						tyInfoData.sProgNm		:= '';
						tyInfoData.udiCode		:= 0;
						tyInfoData.eSeverity	:= AlmSeverityNA;
						tyInfoData.sAlmMsg		:= '';
					ELSE
						IF p_sInfoMsg <> '' THEN
							tyInfoData.sProgNm		:= p_sProgNm;
							tyInfoData.udiCode		:= 10000;
							tyInfoData.eSeverity	:= AlmSeverityInfo;
							tyInfoData.sAlmMsg		:= p_sInfoMsg;
						ELSE
							tyInfoData.sProgNm		:= '';
							tyInfoData.udiCode		:= 0;
							tyInfoData.eSeverity	:= AlmSeverityNA;
							tyInfoData.sAlmMsg		:= '';
						END_IF
					END_IF
				END_IF
			ELSE
				usiProdAccDatStep	:= 6;
			END_IF

		4:
			//Accept New Recipe Name
			IF p_bInternalUse = TRUE THEN

				p_tyCurrProdRcp	:= p_tyInternalReqProdRcp;
				usiProdAccDatStep := 6;
			ELSE

				FOR i := 1 TO 2000 DO
					IF sReqProdRcpNm = '' THEN
						EXIT;
					ELSIF sReqProdRcpNm = pa_tyProdRcpList[i].sRcpNm THEN
						p_tyCurrProdRcp	:= pa_tyProdRcpList[i];

						EXIT;
					END_IF
				END_FOR

				IF i > 2000 THEN
					//Recipe Not Exist
					bProdRcpErr := TRUE;
					bProdRcpErrNotExist	:= TRUE;
				END_IF
				usiProdAccDatStep	:= 5;
			END_IF

		5:
			(* Add *)
			p_tyProdRcpCurrRcpWr 	:= p_tyCurrProdRcp;
			p_eLinkUIProdRcpAct 	:= ProdRcpActWriteCurrRcpParam;

			IF p_eProdRcpStat = ProdRcpActWriteCurrRcpParam AND p_eProdRcpStatus = Done THEN
				p_eLinkUIProdRcpAct := ProdRcpActIdle;
				usiProdAccDatStep := 6;
			END_IF

		6:
			//Clear Info Message
			tyInfoData.sProgNm		:= '';
			tyInfoData.udiCode		:= 0;
			tyInfoData.eSeverity	:= AlmSeverityNA;
			tyInfoData.sAlmMsg		:= '';

			usiProdAccDatStep	:= 0;

	END_CASE

END_ACTION
```

#### Act_Alarm.st - Do Not Change!!!
```iecst
(** 2019-04-21 **)
ACTION Act_Alarm:

	//Error
	IF EDGEPOS(eStatus = Error) THEN

		tyAlmData.sProgNm		:= p_sProgNm;
		tyAlmData.udiCode		:= udiStatus;
		tyAlmData.eSeverity		:= AlmSeverityError;
		tyAlmData.udiRunTime	:= tyAlmData.udiRunTime + 1;
		tyAlmData.bAlm			:= TRUE;
		tyAlmData.udiModuleNum  := udiModuleNum;
		g_sLFFollowerProgNm		:= p_sProgNm;
		//Get Error Message
		IF tyAlmData.udiCode < 10000 OR tyAlmData.udiCode > 10099 THEN
			tyAlmData.sAlmMsg	:= 'Unknown';
			tyAlmData.sRcyMsg	:= 'Unknown';
		ELSE
			tyAlmData.sAlmMsg	:= a_tyAlmText[tyAlmData.udiCode].sAlmText;
			tyAlmData.sRcyMsg	:= a_tyAlmText[tyAlmData.udiCode].sRcyText;
		END_IF

	ELSIF bRstErr AND (tyAlmData.udiCode <> 0) THEN

		tyAlmData.udiCode	:= 0;
		tyAlmData.eSeverity	:= AlmSeverityNA;
		tyAlmData.sAlmMsg	:= '';
		tyAlmData.sRcyMsg	:= '';
		tyAlmData.bAlm			:= FALSE;
	END_IF

END_ACTION
```

#### InputRef.var - Do Not Change!!!
```iecst
(*2020-08-06*)
(**)
(*General*)
VAR
	p_udiRstErr : REFERENCE TO UDINT;
	p_bPrep : REFERENCE TO BOOL;
	p_bEn : REFERENCE TO BOOL;
	p_bDis : REFERENCE TO BOOL;
END_VAR
(**)
(*Configuration*)
VAR
	p_eAWStat : REFERENCE TO eAWAction;
	p_sIPAddr : REFERENCE TO STRING[15];
END_VAR
(**)
(*Input*)
VAR
	p_sMcNm : REFERENCE TO STRING[30];
	p_bAWPrep : REFERENCE TO BOOL;
	p_bAWDis : REFERENCE TO BOOL;
	p_bMnlAccData : REFERENCE TO BOOL;
	p_bSectionLeader : REFERENCE TO BOOL;
	p_sMagRcpNm : REFERENCE TO STRING[30];
	p_diWidthLimit : REFERENCE TO DINT;
	p_bWidth2Prep : REFERENCE TO BOOL;
	p_bUSWidthChkPrep : REFERENCE TO BOOL;
	p_bUSWidthChkEn : REFERENCE TO BOOL;
	p_bUSWidthChkSen : REFERENCE TO BOOL;
	p_bDSWidthChkPrep : REFERENCE TO BOOL;
	p_bDSWidthChkEn : REFERENCE TO BOOL;
	p_bDSWidthChkSen : REFERENCE TO BOOL;
	p_bProdWidthChk : REFERENCE TO BOOL;
	p_bUIProdAccData : REFERENCE TO BOOL;
	p_bUIProdUpdtData : REFERENCE TO BOOL;
	p_bUIMagAccData : REFERENCE TO BOOL;
	pa_tyProdRcpList : REFERENCE TO ARRAY[1..c_udiProdRcpMax] OF tyProdRcpParam;
	p_tyCurrProdRcp : REFERENCE TO tyProdRcpParam;
	p_sCurrMagRcpNm : REFERENCE TO STRING[30];
	p_eTimeStat : REFERENCE TO eTimeAction;
	p_eTimeStatus : REFERENCE TO eFBStatus;
	p_bAccNewRcpCond : REFERENCE TO BOOL;
	p_bUpdtNewRcpCond : REFERENCE TO BOOL;
	p_bAutoUpdtData : REFERENCE TO BOOL;
	p_sInfoMsg : REFERENCE TO STRING[200];
	p_bInternalUse : REFERENCE TO BOOL;
	p_tyInternalReqProdRcp : REFERENCE TO tyProdRcpParam;
	p_bNewBrdEnteredCond : REFERENCE TO BOOL;
	p_bOldBrdExitedCond : REFERENCE TO BOOL;
	p_bRlsBrd : REFERENCE TO BOOL;
	p_tyToLeaderProdRcp : REFERENCE TO tyProdRcpParam;
	p_bInternalReqProdRcpDiff : REFERENCE TO BOOL;
	p_bUpdtProdRcpDiff : REFERENCE TO BOOL;
	p_bRlsBrdProdRcpDiff : REFERENCE TO BOOL;
	p_sProgNm : REFERENCE TO STRING[15];
	p_bNtSettingsLoadDone : REFERENCE TO BOOL;
	p_tOnlineChkDlyTm : REFERENCE TO TIME;
	p_bManual : REFERENCE TO BOOL;
	p_bErr : REFERENCE TO BOOL;
	p_bWarning : REFERENCE TO BOOL;
	p_bOps : REFERENCE TO BOOL;
	p_bStandby : REFERENCE TO BOOL;
	p_bDBAOnWOAlign : REFERENCE TO BOOL;
END_VAR
```

#### Local.var - Do Not Change!!!
```iecst
(*2021-05-18*)
(**)
(*Local Action, State & Status*)
VAR
	eStatus : eFBStatus := Idle;
	udiStatus : UDINT := 0;
END_VAR
(**)
(*Local Alarm*)
VAR
	tyAlmData : tyAlmDat;
	tyInfoData : tyAlmDat;
	tyInfoData1 : tyAlmDat;
	a_tyAlmText : ARRAY[10000..10099] OF tyAlmTxt := [(sAlmText:='New Recipe Not Found In Product Recipe List',sRcyText:='Create New Recipe In Product Setting.'),(sAlmText:='Product Recipe Width Not Match',sRcyText:='Check Product Width And Leader Request Width'),(sAlmText:='New Recipe Not Found In Magazine Recipe List',sRcyText:='Create New Recipe In Magazine Setting.'),(sAlmText:='New Recipe Name Empty',sRcyText:='Request Recipe Name From Leader Is Empty, Check Leader Machine'),96(0)];
END_VAR
(**)
(*Local Output*)
VAR
	bUSAllow : BOOL;
	bDSAllow : BOOL;
	bLeaderSeqCtrlInActive : BOOL;
	bProdAccDataMnl : BOOL;
	bProdUpdtDataMnl : BOOL;
	bMagAccDataMnl : BOOL;
	eTimeAct : eTimeAction;
	bWaitRlsBrd : BOOL;
	tyLeaderInfo : tyLFLeaderInfo;
	tyUpdtProdRcp : tyProdRcpParam;
END_VAR
(**)
(*Local Input*)
VAR
	udiRstErr : UDINT := 0;
	bPrep : BOOL := TRUE;
	bEn : BOOL := TRUE;
	bDis : BOOL := FALSE;
	sIPAddr : STRING[15] := '192.168.0.100';
	sMcNm : STRING[30];
	bAWPrep : BOOL := TRUE;
	bAWDis : BOOL;
	bMnlAccData : BOOL;
	bSectionLeader : BOOL;
	sMagRcpNm : STRING[30];
	diWidthLimit : DINT;
	bWidth2Prep : BOOL;
	bUSWidthChkPrep : BOOL;
	bUSWidthChkEn : BOOL;
	bUSWidthChkSen : BOOL;
	bDSWidthChkPrep : BOOL;
	bDSWidthChkEn : BOOL;
	bDSWidthChkSen : BOOL;
	bProdWidthChk : BOOL;
	bUIProdAccData : BOOL;
	bUIProdUpdtData : BOOL;
	bUIMagAccData : BOOL;
	a_tyProdRcpList : ARRAY[1..c_udiProdRcpMax] OF tyProdRcpParam;
	tyCurrProdRcp : tyProdRcpParam;
	sCurrMagRcpNm : STRING[30];
	eTimeStat : eTimeAction;
	eTimeStatus : eFBStatus;
	bAccNewRcpCond : BOOL;
	bUpdtNewRcpCond : BOOL;
	bAutoUpdtData : BOOL;
	sInfoMsg : STRING[200];
	bInternalUse : BOOL;
	tyInternalReqProdRcp : tyProdRcpParam;
	bNewBrdEnteredCond : BOOL;
	bOldBrdExitedCond : BOOL;
	bRlsBrd : BOOL;
	tyToLeaderProdRcp : tyProdRcpParam;
	bInternalReqProdRcpDiff : BOOL;
	bUpdtProdRcpDiff : BOOL;
	bRlsBrdProdRcpDiff : BOOL;
	sProgNm : STRING[15] := 'Follower';
	bNtSettingsLoadDone : BOOL := TRUE;
	tOnlineChkDlyTm : TIME;
	bManual : BOOL := FALSE;
	bErr : BOOL := FALSE;
	bWarning : BOOL := FALSE;
	bOps : BOOL := FALSE;
	bStandby : BOOL := FALSE;
	eAWStat : eAWAction;
END_VAR
(**)
(*Local*)
VAR
	bRstErr : BOOL;
	udiRstErrOld : UDINT;
	bInitDone : BOOL;
	bInitialDone : BOOL;
	bAutoAccData : BOOL;
	bProdRcpErr : BOOL;
	bMagRcpErr : BOOL;
	bSetTmErr : BOOL;
	bProdAccDataReq : BOOL;
	sReqProdRcpNm : STRING[254];
	diReqProdRcpWidth : DINT;
	bMagAccDataReq : BOOL;
	sReqMagRcpNm : STRING[30];
	usiProdAccDatStep : USINT;
	usiMagAccDatStep : USINT;
	usiProdUpdtDatStep : USINT;
	tyRlsBrdProdRcpNm : tyProdRcpParam;
	bNewBrdEntered : BOOL;
	bOldBrdExited : BOOL;
	i : INT;
	bSetTm : BOOL;
	fbOnlineChk : fbLFFollowerOnlineChk;
	fbFollower : fbLFFollower;
	tyLeaderToFollowerTag : tyLFLeaderToFollowerTag;
	tyFollowerToLeaderTag : tyLFFollowerToLeaderTag;
	eCurrMachineStat : eMachineStat;
	bLeaderOnline : BOOL;
	bLeaderInfo : BOOL;
	bFollowerInfo : BOOL;
	bProdRcpErrNotExist : BOOL;
	bProdRcpErrWidthMismatch : BOOL;
	bDBAOnWOAlign : BOOL;
	udiModuleNum : UDINT := 3901;
END_VAR
```

### LCS.typ - Change By Project
```iecst
(*2019-07-10*)
(**)
(*Action*)

TYPE
	eLCSAction :
		(
		LCSActIdle := 0,
		LCSActAddProd := 1,
		LCSActAddMultiProd := 2,
		LCSActEditProd := 3,
		LCSActEditMultiProd := 4,
		LCSActOverWriteProd := 5,
		LCSActOverWriteMultiProd := 6,
		LCSActDelProd := 7,
		LCSActDelMultiProd := 8,
		LCSActRunProd := 9,
		LCSActUploadProd := 10,
		LCSActUploadMultiProd := 11
		);
END_TYPE

(**)
(*Data*)

TYPE
	eLCSOpsStatus :
		(
		LCSOpsStatusAuto,
		LCSOpsStatusManual,
		LCSOpsStatusStop,
		LCSOpsStatusError,
		LCSOpsStatusWarning
		);
	tyLCSTagNm : 	STRUCT
		eAct : eLCSAction;
		eStat : eLCSAction;
		udiStatus : UDINT;
		sErrMsg : STRING[200];
		iIdxAct : INT;
		iIdxStat : INT;
		tyProdRcpInfo : tyProdRcpParam;
		tyCurrProdRcpParam : tyProdRcpParam;
		sCurrRcpNm : STRING[30];
		rCurrWidth : REAL;
		eCurrOpsStatus : eLCSOpsStatus;
		usiBrdStatus : USINT;
		usiMode : USINT;
		sLastModified : STRING[80];
		bMngRcpEn : BOOL;
		bLiveData : BOOL;
		bLFEn : BOOL;
		sMcAlmMsg : ARRAY[1..c_udiAlarmCurrMax]OF STRING[255];
		bSectionLeaderEn : BOOL;
	END_STRUCT;
END_TYPE
```

### LCS.var - Change By Project
```iecst
(*2019-04-24*)
(**)
(*Action & State & Status*)
(**)
(*Alarm*)
(**)
(*Output*)
VAR
	p_LCS_LCSMngRcp_LCSAct : UDINT;
	p_LCS_LCSMngRcp_LCSIdxAct : UDINT;
	p_LCS_LCSMngRcp_LCSIdxStat : UDINT;
	p_LCS_LCSMngRcp_LCSProdRcpInfo : UDINT;
	p_LCS_LCSLF_LCSAct : UDINT;
	p_LCS_LCSLF_LCSProdRcpInfo : UDINT;
	p_LCSChkLmtOK : UDINT;
	p_LCSChkLmtNG : UDINT;
	p_LCSSectionLeaderEn : UDINT;
END_VAR
```

### Program Logical/LCS/LCS (IEC, version 1.00.0) - 1.00.0 - NtRecipe v5.00.0 , NtFileIO v5.00.0

#### Init.st - Change By Project
```iecst
(** 2019-04-24 **)
PROGRAM _INIT

	(* Always Change If Project Change *)

	//Pass Address To Global Address For External Use
	//Action, State & Status

	//Alarm

	//Output
	p_LCS_LCSMngRcp_LCSAct			:= ADR(eLCSMngRcp_LCSAct);
	p_LCS_LCSMngRcp_LCSIdxAct		:= ADR(iLCSMngRcp_LCSIdxAct);
	p_LCS_LCSMngRcp_LCSIdxStat		:= ADR(iLCSMngRcp_LCSIdxStat);
	p_LCS_LCSMngRcp_LCSProdRcpInfo	:= ADR(tyLCSMngRcp_LCSProdRcpInfo);
	p_LCS_LCSLF_LCSAct				:= ADR(eLCSLF_LCSAct);
	p_LCS_LCSLF_LCSProdRcpInfo		:= ADR(tyLCSLF_LCSProdRcpInfo);
	p_LCSChkLmtOK					:= ADR(bChkLmtOK);
	p_LCSChkLmtNG					:= ADR(bChkLmtNG);
	p_LCSSectionLeaderEn			:= ADR(tyTagNm.bSectionLeaderEn);

	(* Always Change If Project Change *)

END_PROGRAM
```

#### Act_InitGlobal.st - Change By Project
```iecst
(** 2019-06-12 **)
ACTION Act_InitGlobal:

	(* Always Change If Project Change *)

	//Pass Data To Link
	p_bLinkStartupRun ACCESS p_StartupRun;
	p_bLinkNtParamLCSLFPrep ACCESS p_NtParamLCSLFPrep;
	p_bLinkNtParamLCSManageRcpPrep ACCESS p_NtParamLCSManageRcpPrep;
	p_bLinkNtParamLCSReqRcpPrep ACCESS p_NtParamLCSReqRcpPrep;
	p_bLinkNtParamLCSLiveDatPrep ACCESS p_NtParamLCSLiveDatPrep;
	p_bLinkMcParamLCSLFEn ACCESS p_McParamLCSLFEn;
	p_bLinkMcParamLCSManageRcpEn ACCESS p_McParamLCSManageRcpEn;
	p_bLinkMcParamLCSReqRcpEn ACCESS p_McParamLCSReqRcpEn;
	p_bLinkMcParamLCSLiveDatEn ACCESS p_McParamLCSLiveDatEn;
	p_tyLinkUpdtProdRcp ACCESS p_Follower1UpdtProdRcp;

	p_bLinkConvHvBrd ACCESS p_OpsInvertHvBrd;
	p_tyLinkAlarmCurrList ACCESS p_AlarmCurrList;

	//Pass Data To Internal Use
	p_eLCSMngRcp_PLCStat ACCESS p_LCSMngRcpStat;
	p_udiLCSMngRcp_PLCStatus ACCESS p_LCSMngRcp_PLCStatus;
	p_iLCSMngRcp_PLCIdxAct ACCESS p_LCSMngRcp_PLCIdxAct;
	p_iLCSMngRcp_PLCIdxStat ACCESS p_LCSMngRcp_PLCIdxStat;
	p_tyLCSMngRcp_PLCProdRcpInfo ACCESS p_LCSMngRcp_PLCProdRcpInfo;
	p_eLCSLF_PLCStat ACCESS p_LCSLFStat;
	p_udiLCSLF_PLCStatus ACCESS p_LCSLF_PLCStatus;
	p_bLCSMngRcpChkLmt ACCESS p_LCSMngRcpChkLmt;
	p_bLCSLFChkLmt ACCESS p_LCSLFChkLmt;
	p_bOpsRun ACCESS p_OpsRun;
	p_bError ACCESS p_AlarmErr;
	p_bWarning ACCESS p_AlarmWarning;
	p_bInfo ACCESS p_AlarmInfo;
	p_bUIManual ACCESS p_UIUIMnlMod;
	p_tyProdRcpCurrRcp ACCESS p_Follower1UpdtProdRcp;	//Assign With Conveyor Last Zone (Live Data Update)
	p_tyNtParamCurr ACCESS p_NtParamCurr;
	p_sProgNm ACCESS p_NtParamLCSProgNm;
	p_bNtSettingsLoadDone ACCESS p_StartupNtSettingsLoadDone;

	(* Always Change If Project Change *)

END_ACTION
```

#### InputRef_Link.var - Change By Project
```iecst
(*2019-04-24*)
(**)
VAR
	p_bLinkStartupRun : REFERENCE TO BOOL;
	p_bLinkNtParamLCSLFPrep : REFERENCE TO BOOL;
	p_bLinkNtParamLCSManageRcpPrep : REFERENCE TO BOOL;
	p_bLinkNtParamLCSReqRcpPrep : REFERENCE TO BOOL;
	p_bLinkNtParamLCSLiveDatPrep : REFERENCE TO BOOL;
	p_bLinkMcParamLCSLFEn : REFERENCE TO BOOL;
	p_bLinkMcParamLCSManageRcpEn : REFERENCE TO BOOL;
	p_bLinkMcParamLCSReqRcpEn : REFERENCE TO BOOL;
	p_bLinkMcParamLCSLiveDatEn : REFERENCE TO BOOL;
	p_tyLinkUpdtProdRcp : REFERENCE TO tyProdRcpParam;
	p_sLinkUpdtProdRcpNm : REFERENCE TO STRING[30];
	p_diLinkUpdtProdWidth : REFERENCE TO DINT;
END_VAR
(**)
VAR
	p_bLinkConvHvBrd : REFERENCE TO BOOL;
	p_tyLinkAlarmCurrList : REFERENCE TO ARRAY[1..c_udiAlarmCurrMax] OF tyAlarmCurr;
END_VAR
```

#### Act_LinkEn.st - Change By Project
```iecst
(** 2019-04-24 **)
ACTION Act_LinkEn:

	//Link bPrep, bEn & bDis
	p_bPrep	:= p_bLinkNtParamLCSLFPrep OR p_bLinkNtParamLCSManageRcpPrep OR p_bLinkNtParamLCSReqRcpPrep OR p_bLinkNtParamLCSLiveDatPrep;
	p_bEn	:= p_bLinkMcParamLCSLFEn OR p_bLinkMcParamLCSManageRcpEn OR p_bLinkMcParamLCSReqRcpEn OR p_bLinkMcParamLCSLiveDatEn;
	p_bDis	:= p_bLinkStartupRun;

END_ACTION
```

#### Act_Link.st - Change By Project
```iecst
(** 2019-07-10 **)
ACTION Act_Link:

	//Check Limit
	IF p_bLCSMngRcpChkLmt OR p_bLCSLFChkLmt THEN

		IF tyTagNm.tyProdRcpInfo.sRcpNm = '' THEN

			bChkLmtOK	:= FALSE;
			bChkLmtNG	:= TRUE;
			sAddMsg		:= 'Recipe Name Empty ';

		ELSIF tyTagNm.tyProdRcpInfo.diWidthInUM < p_tyNtParamCurr.tyProdRcpWidthLmt.diMin THEN

			bChkLmtOK	:= FALSE;
			bChkLmtNG	:= TRUE;
			sAddMsg		:= 'Width Lower Limit ';

		ELSIF tyTagNm.tyProdRcpInfo.diWidthInUM > p_tyNtParamCurr.tyProdRcpWidthLmt.diMax THEN

			bChkLmtOK	:= FALSE;
			bChkLmtNG	:= TRUE;
			sAddMsg		:= 'Width Upper Limit ';
		ELSIF tyTagNm.tyProdRcpInfo.usiMcMod < DINT_TO_USINT(p_tyNtParamCurr.tyProdRcpMcModLmt.diMin) THEN

			bChkLmtOK	:= FALSE;
			bChkLmtNG	:= TRUE;
			sAddMsg		:= 'Machine Mode Lower Limit ';

		ELSIF tyTagNm.tyProdRcpInfo.usiMcMod > DINT_TO_USINT(p_tyNtParamCurr.tyProdRcpMcModLmt.diMax) THEN

			bChkLmtOK	:= FALSE;
			bChkLmtNG	:= TRUE;
			sAddMsg		:= 'Machine Mode Upper Limit ';

		ELSE

			bChkLmtOK	:= TRUE;
			bChkLmtNG	:= FALSE;
			sAddMsg		:= '';

		END_IF

	ELSE

		bChkLmtOK	:= FALSE;
		bChkLmtNG	:= FALSE;

	END_IF

	//Update LCS Enable
	tyTagNm.bMngRcpEn		:= p_bLinkNtParamLCSManageRcpPrep AND p_bLinkMcParamLCSManageRcpEn;
	tyTagNm.bLFEn			:= p_bLinkNtParamLCSLFPrep AND p_bLinkMcParamLCSLFEn;
	tyTagNm.bLiveData		:= p_bLinkNtParamLCSLiveDatPrep AND p_bLinkMcParamLCSLiveDatEn;
	tyTagNm.usiBrdStatus	:= BOOL_TO_USINT(p_bLinkConvHvBrd);

	//Action
	IF tyTagNm.eAct = LCSActRunProd THEN

		bLFRun		:= TRUE;
		bMngRcpRun	:= FALSE;

	ELSIF (tyTagNm.eAct = LCSActAddProd)
		OR (tyTagNm.eAct = LCSActAddMultiProd)
		OR (tyTagNm.eAct = LCSActEditProd)
		OR (tyTagNm.eAct = LCSActEditMultiProd)
		OR (tyTagNm.eAct = LCSActOverWriteProd)
		OR (tyTagNm.eAct = LCSActOverWriteMultiProd)
		OR (tyTagNm.eAct = LCSActDelProd)
		OR (tyTagNm.eAct = LCSActDelMultiProd)
		OR (tyTagNm.eAct = LCSActUploadProd)
		OR (tyTagNm.eAct = LCSActUploadMultiProd) THEN

		bLFRun		:= FALSE;
		bMngRcpRun	:= TRUE;

	ELSIF tyTagNm.eAct = LCSActIdle THEN

		bLFRun		:= FALSE;
		bMngRcpRun	:= FALSE;

	END_IF

	IF bLFRun = TRUE THEN
		eLCSLF_LCSAct			:= tyTagNm.eAct;
		tyLCSLF_LCSProdRcpInfo	:= tyTagNm.tyProdRcpInfo;

		sLastModifiedTemp	:= CONCAT('DT#' , tyTagNm.sLastModified);
		tyLCSLF_LCSProdRcpInfo.dtLastModified	:= STRING_TO_DT(sLastModifiedTemp);

		tyTagNm.eStat		:= p_eLCSLF_PLCStat;
		tyTagNm.udiStatus	:= p_udiLCSLF_PLCStatus;

		IF tyTagNm.udiStatus > 0 AND tyTagNm.udiStatus < 65534 THEN
			tyTagNm.sErrMsg	:= a_tyAlmText[tyTagNm.udiStatus].sAlmText;

			IF tyTagNm.udiStatus = 10010 OR tyTagNm.udiStatus = 10011 THEN
				tyTagNm.sErrMsg	:= CONCAT(sAddMsg , tyTagNm.sErrMsg);
			END_IF
		END_IF

	ELSIF bMngRcpRun = TRUE THEN
		eLCSMngRcp_LCSAct	:= tyTagNm.eAct;

		tyTagNm.eStat		:= p_eLCSMngRcp_PLCStat;
		tyTagNm.udiStatus	:= p_udiLCSMngRcp_PLCStatus;

		IF tyTagNm.udiStatus > 0 AND tyTagNm.udiStatus < 65534 THEN
			tyTagNm.sErrMsg	:= a_tyAlmText[tyTagNm.udiStatus].sAlmText;

			IF tyTagNm.udiStatus = 10010 OR tyTagNm.udiStatus = 10011 THEN
				tyTagNm.sErrMsg	:= CONCAT(sAddMsg , tyTagNm.sErrMsg);
			END_IF
		END_IF

		IF tyTagNm.eAct = LCSActUploadProd THEN
			IF tyTagNm.udiStatus = 0 THEN
				tyTagNm.tyProdRcpInfo	:= p_tyLCSMngRcp_PLCProdRcpInfo;

				tyTagNm.sLastModified	:= DT_TO_STRING(tyLCSMngRcp_LCSProdRcpInfo.dtLastModified);
				tyTagNm.sLastModified	:= RIGHT(tyTagNm.sLastModified , (LEN(tyTagNm.sLastModified) - 3));

			ELSE
				tyLCSMngRcp_LCSProdRcpInfo	:= tyTagNm.tyProdRcpInfo;

				tyLCSMngRcp_LCSProdRcpInfo.diWidthInUM2 := tyTagNm.tyProdRcpInfo.diWidthInUM; //Added

				sLastModifiedTemp	:= CONCAT('DT#' , tyTagNm.sLastModified);
				tyLCSMngRcp_LCSProdRcpInfo.dtLastModified	:= STRING_TO_DT(sLastModifiedTemp);

			END_IF

		ELSIF tyTagNm.eAct = LCSActUploadMultiProd THEN
			iLCSMngRcp_LCSIdxStat	:= tyTagNm.iIdxAct;

			tyTagNm.iIdxStat		:= p_iLCSMngRcp_PLCIdxAct;

			tyTagNm.tyProdRcpInfo	:= p_tyLCSMngRcp_PLCProdRcpInfo;

			tyTagNm.sLastModified	:= DT_TO_STRING(tyLCSMngRcp_LCSProdRcpInfo.dtLastModified);
			tyTagNm.sLastModified	:= RIGHT(tyTagNm.sLastModified , (LEN(tyTagNm.sLastModified) - 3));

		ELSE
			iLCSMngRcp_LCSIdxAct		:= tyTagNm.iIdxAct;
			tyLCSMngRcp_LCSProdRcpInfo	:= tyTagNm.tyProdRcpInfo;

			tyLCSMngRcp_LCSProdRcpInfo.diWidthInUM2 := tyTagNm.tyProdRcpInfo.diWidthInUM; //Added

			sLastModifiedTemp	:= CONCAT('DT#' , tyTagNm.sLastModified);
			tyLCSMngRcp_LCSProdRcpInfo.dtLastModified	:= STRING_TO_DT(sLastModifiedTemp);

			tyTagNm.iIdxStat	:= p_iLCSMngRcp_PLCIdxStat;

		END_IF

	ELSE

		eLCSLF_LCSAct		:= LCSActIdle;
		eLCSMngRcp_LCSAct	:= LCSActIdle;
		tyTagNm.eStat		:= LCSActIdle;
		tyTagNm.udiStatus	:= 65534;
		tyTagNm.sErrMsg		:= '';

	END_IF

END_ACTION
```

#### Cyclic.st - Do Not Change!!!
```iecst
(** 2019-04-30 **)
PROGRAM _CYCLIC

	IF bInitDone = FALSE THEN
		bInitDone	:= TRUE;

		Act_InitLocal;
		Act_InitGlobal;

	ELSIF bInitialDone = FALSE THEN
		IF p_bNtSettingsLoadDone = TRUE THEN
			bInitialDone	:= TRUE;

			Act_Initial;
		END_IF

	ELSE

		Act_LinkEn;

		IF (p_bPrep = TRUE) AND (p_bEn = TRUE) AND (p_bDis = FALSE) THEN
			Act_Link;
			Act_Background;
		ELSE
			Act_Main_Disable;

			tyTagNm.udiStatus	:= 10000;	//LCS Disable
		END_IF

	END_IF

END_PROGRAM
```

#### Act_InitLocal.st - Do Not Change!!!
```iecst
(** 2019-06-12 **)
ACTION Act_InitLocal:

	//Input Reference Link To Local Variable
	p_bPrep ACCESS ADR(bPrep);
	p_bEn ACCESS ADR(bEn);
	p_bDis ACCESS ADR(bDis);
	p_eLCSMngRcp_PLCStat ACCESS ADR(eLCSMngRcp_PLCStat);
	p_udiLCSMngRcp_PLCStatus ACCESS ADR(udiLCSMngRcp_PLCStatus);
	p_iLCSMngRcp_PLCIdxAct ACCESS ADR(iLCSMngRcp_PLCIdxAct);
	p_iLCSMngRcp_PLCIdxStat ACCESS ADR(iLCSMngRcp_PLCIdxStat);
	p_tyLCSMngRcp_PLCProdRcpInfo ACCESS ADR(tyLCSMngRcp_PLCProdRcpInfo);
	p_eLCSLF_PLCStat ACCESS ADR(eLCSLF_PLCStat);
	p_udiLCSLF_PLCStatus ACCESS ADR(udiLCSLF_PLCStatus);
	p_bLCSMngRcpChkLmt ACCESS ADR(bLCSMngRcpChkLmt);
	p_bLCSLFChkLmt ACCESS ADR(bLCSLFChkLmt);
	p_bOpsRun ACCESS ADR(bOpsRun);
	p_bError ACCESS ADR(bError);
	p_bWarning ACCESS ADR(bWarning);
	p_bInfo ACCESS ADR(bInfo);
	p_bUIManual ACCESS ADR(bUIManual);
	p_tyProdRcpCurrRcp ACCESS ADR(tyProdRcpCurrRcp);
	p_tyNtParamCurr ACCESS ADR(tyNtParamCurr);
	p_sProgNm ACCESS ADR(sProgNm);
	p_bNtSettingsLoadDone ACCESS ADR(bNtSettingsLoadDone);

END_ACTION
```

#### Act_Initial.st - Do Not Change!!!
```iecst
(** 2019-04-24 **)
ACTION Act_Initial:

	//Initial

END_ACTION
```

#### Act_Background.st - Do Not Change!!!
```iecst
(** 2019-05-21 **)
ACTION Act_Background:

	Act_Background_LiveData;

	IF udiFlagNo = 0 THEN
		memset(ADR(tyTagNm.sMcAlmMsg),0,SIZEOF(tyTagNm.sMcAlmMsg));
		FOR udi := 1 TO c_udiAlarmCurrMax DO
			IF 	p_tyLinkAlarmCurrList[udi].sMsg <> '' THEN
				tyTagNm.sMcAlmMsg[udi] := p_tyLinkAlarmCurrList[udi].sMsg;
			ELSIF udi =1 THEN
				EXIT;
			ELSE
				udiFlagNo := udi;
				EXIT;
			END_IF
		END_FOR
	ELSE //For additional alarm occur
		FOR udi := 1 TO c_udiAlarmCurrMax DO
			IF 	p_tyLinkAlarmCurrList[udi].sMsg <> '' THEN
			ELSE
				IF udiFlagNo <> udi THEN
					udiFlagNo := 0;
				END_IF
				EXIT;
			END_IF
		END_FOR
	END_IF

	IF EDGENEG(p_bError) THEN
		udiFlagNo := 0;
		memset(ADR(tyTagNm.sMcAlmMsg),0,SIZEOF(tyTagNm.sMcAlmMsg));
	END_IF

END_ACTION
```

#### Act_Background_LiveData.st - Do Not Change!!!
```iecst
(** 2019-07-10 **)
ACTION Act_Background_LiveData:

	IF p_bLinkNtParamLCSLiveDatPrep AND p_bLinkMcParamLCSLiveDatEn THEN

		tyTagNm.sCurrRcpNm	:= p_tyProdRcpCurrRcp.sRcpNm;
		tyTagNm.rCurrWidth	:= DINT_TO_REAL(p_tyProdRcpCurrRcp.diWidthInUM) / 1000;
		tyTagNm.usiMode		:= BOOL_TO_USINT(p_bLinkNtParamLCSLFPrep AND p_bLinkMcParamLCSLFEn);

		IF p_bError = TRUE THEN
			tyTagNm.eCurrOpsStatus	:= LCSOpsStatusError;
		ELSIF p_bWarning = TRUE OR p_bInfo = TRUE THEN
			tyTagNm.eCurrOpsStatus	:= LCSOpsStatusWarning;
		ELSIF p_bOpsRun = TRUE THEN
			tyTagNm.eCurrOpsStatus	:= LCSOpsStatusAuto;
		ELSIF p_bUIManual = TRUE THEN
			tyTagNm.eCurrOpsStatus	:= LCSOpsStatusManual;
		ELSE
			tyTagNm.eCurrOpsStatus	:= LCSOpsStatusStop;
		END_IF

	END_IF

END_ACTION
```

#### Act_Main_Disable.st - Do Not Change!!!
```iecst
(** 2019-04-24 **)
ACTION Act_Main_Disable:

END_ACTION
```

#### InputRef.var - Do Not Change!!!
```iecst
(*2019-06-12*)
(**)
(*General*)
VAR
	p_bPrep : REFERENCE TO BOOL;
	p_bEn : REFERENCE TO BOOL;
	p_bDis : REFERENCE TO BOOL;
END_VAR
(**)
(*Configuration*)
VAR
	p_eLCSMngRcp_PLCStat : REFERENCE TO eLCSAction;
	p_udiLCSMngRcp_PLCStatus : REFERENCE TO UDINT;
	p_iLCSMngRcp_PLCIdxAct : REFERENCE TO INT;
	p_iLCSMngRcp_PLCIdxStat : REFERENCE TO INT;
	p_tyLCSMngRcp_PLCProdRcpInfo : REFERENCE TO tyProdRcpParam;
	p_eLCSLF_PLCStat : REFERENCE TO eLCSAction;
	p_udiLCSLF_PLCStatus : REFERENCE TO UDINT;
	p_bLCSMngRcpChkLmt : REFERENCE TO BOOL;
	p_bLCSLFChkLmt : REFERENCE TO BOOL;
	p_bOpsRun : REFERENCE TO BOOL;
	p_bError : REFERENCE TO BOOL;
	p_bWarning : REFERENCE TO BOOL;
	p_bInfo : REFERENCE TO BOOL;
	p_bUIManual : REFERENCE TO BOOL;
	p_tyProdRcpCurrRcp : REFERENCE TO tyProdRcpParam;
	p_tyNtParamCurr : REFERENCE TO tyNtParam;
	p_sProgNm : REFERENCE TO STRING[15];
	p_bNtSettingsLoadDone : REFERENCE TO BOOL;
END_VAR
```

#### Local.var - Do Not Change!!!
```iecst
(*2019-06-12*)
(**)
(*Local Action, State & Status*)
(**)
(*Local Alarm*)
VAR
	a_tyAlmText : ARRAY[10000..10099] OF tyAlmTxt := [(sAlmText:='LCS Disable'),(sAlmText:='LCS Manage Recipe Disabled'),(sAlmText:='LCS Leader Follower Disabled'),7(0),(sAlmText:='Out Of Range While Accepting New Recipe'),(sAlmText:='Out Of Range While Managing Product'),(sAlmText:='Recipe Name Empty While Adding Product'),(sAlmText:='Recipe List Full While Adding Product'),(sAlmText:='Recipe Name Exist While Adding Product'),(sAlmText:='Recipe Program Error While Adding Product'),(sAlmText:='Check Limit Error While Adding Multiple Product'),(sAlmText:='Recipe Name Empty While Adding Multiple Product'),(sAlmText:='Recipe List Full While Adding Multiple Product'),(sAlmText:='Recipe Name Exist While Adding Multiple Product'),(sAlmText:='Recipe Program Error While Adding Multiple Product'),(sAlmText:='Check Limit Error While Editing Product'),(sAlmText:='Recipe Name Empty While Editing Product'),(sAlmText:='Recipe Name Not Exist While Editing Product'),(sAlmText:='Recipe Program Error While Editing Product'),(sAlmText:='Check Limit Error While Editing Multiple Product'),(sAlmText:='Recipe Name Empty While Editing Multiple Product'),(sAlmText:='Recipe Name Not Exist While Editing Multiple Product'),(sAlmText:='Recipe Program Error While Editing Multiple Product'),(sAlmText:='Check Limit Error While Overwriting Product'),(sAlmText:='Recipe Name Empty While Overwriting Product'),(sAlmText:='Recipe List Full While Overwriting Product'),(sAlmText:='Recipe Program Error While Overwriting Product'),(sAlmText:='Check Limit Error While Overwriting Multiple Product'),(sAlmText:='Recipe Name Empty While Overwriting Multiple Product'),(sAlmText:='Recipe List Full While Overwriting Multiple Product'),(sAlmText:='Recipe Program Error While Overwriting Multiple Product'),(sAlmText:='Check Limit Error While Deleting Product'),(sAlmText:='Recipe Name Empty While Deleting Product'),(sAlmText:='Recipe Name Not Exist While Deleting Product'),(sAlmText:='Recipe Program Error While Deleting Product'),(sAlmText:='Check Limit Error While Deleting Multiple Product'),(sAlmText:='Recipe Name Empty While Deleting Multiple Product'),(sAlmText:='Recipe Name Not Exist While Deleting Multiple Product'),(sAlmText:='Recipe Program Error While Deleting Multiple Product'),(sAlmText:='Recipe Name Empty While Uploading Product'),(sAlmText:='Recipe Name Not Exist While Uploading Product'),(sAlmText:='Recipe Program Error While Uploading Product'),(sAlmText:='Get Recipe Info Error While Editing Product'),(sAlmText:='Local Recipe Is Latest Compare With LCS Recipe While Editing Product'),(sAlmText:='Local Recipe Is Latest Compare With LCS Recipe While Editing Multiple Product'),(sAlmText:='Get Recipe Info Error While Editing Multiple Product'),48(0)];
END_VAR
(**)
(*Local Output*)
VAR
	eLCSMngRcp_LCSAct : eLCSAction;
	iLCSMngRcp_LCSIdxAct : INT;
	iLCSMngRcp_LCSIdxStat : INT;
	tyLCSMngRcp_LCSProdRcpInfo : tyProdRcpParam;
	eLCSLF_LCSAct : eLCSAction;
	tyLCSLF_LCSProdRcpInfo : tyProdRcpParam;
	bChkLmtOK : BOOL;
	bChkLmtNG : BOOL;
END_VAR
(**)
(*Local Input*)
VAR
	bPrep : BOOL := TRUE;
	bEn : BOOL := TRUE;
	bDis : BOOL := FALSE;
	eLCSMngRcp_PLCStat : eLCSAction;
	udiLCSMngRcp_PLCStatus : UDINT;
	iLCSMngRcp_PLCIdxAct : INT;
	iLCSMngRcp_PLCIdxStat : INT;
	tyLCSMngRcp_PLCProdRcpInfo : tyProdRcpParam;
	eLCSLF_PLCStat : eLCSAction;
	udiLCSLF_PLCStatus : UDINT;
	bLCSMngRcpChkLmt : BOOL;
	bLCSLFChkLmt : BOOL;
	bOpsRun : BOOL;
	bError : BOOL;
	bWarning : BOOL;
	bInfo : BOOL;
	bUIManual : BOOL;
	tyProdRcpCurrRcp : tyProdRcpParam;
	tyNtParamCurr : tyNtParam;
	sProgNm : STRING[15] := 'LCS';
	bNtSettingsLoadDone : BOOL := TRUE;
END_VAR
(**)
(*Local*)
VAR
	udi : UDINT;
	udiFlagNo : UDINT;
	bInitDone : BOOL;
	bInitialDone : BOOL;
	tyTagNm : tyLCSTagNm;
	bLFRun : BOOL;
	bMngRcpRun : BOOL;
	sLastModifiedTemp : STRING[80];
	sAddMsg : STRING[80];
	udiModuleNum : UDINT := 4001;
END_VAR
```

### LCSMngRcp.var - Change By Project
```iecst
(*2019-04-24*)
(**)
(*Action & State & Status*)
VAR
	p_LCSMngRcpStat : UDINT;
	p_LCSMngRcpStatus : UDINT;
	p_LCSMngRcpStatTxt : UDINT;
END_VAR
(**)
(*Alarm*)
VAR
	p_LCSMngRcpAlmData : UDINT;
END_VAR
(**)
(*Output*)
VAR
	p_LCSMngRcp_PLCStatus : UDINT;
	p_LCSMngRcp_PLCIdxAct : UDINT;
	p_LCSMngRcp_PLCIdxStat : UDINT;
	p_LCSMngRcp_PLCProdRcpInfo : UDINT;
	p_LCSMngRcpProdRcpAct : UDINT;
	p_LCSMngRcpProdRcpInfoIn : UDINT;
	p_LCSMngRcpChkLmt : UDINT;
END_VAR
```

### Program Logical/LCS/LCSMngRcp (IEC, version 1.00.0) - 1.00.0 - NtRecipe v5.00.0 , NtFileIO v5.00.0

#### Init.st - Change By Project
```iecst
(** 2019-04-24 **)
PROGRAM _INIT

	(* Always Change If Project Change *)

	//Pass Address To Global Address For External Use
	//Action, State & Status
	p_LCSMngRcpStat		:= ADR(eStat);
	p_LCSMngRcpStatus	:= ADR(eStatus);
	p_LCSMngRcpStatTxt	:= ADR(sStatTxt);

	//Alarm
	p_LCSMngRcpAlmData	:= ADR(tyAlmData);

	//Output
	p_LCSMngRcp_PLCStatus		:= ADR(udiPLCStatus);
	p_LCSMngRcp_PLCIdxAct		:= ADR(iPLCIdxAct);
	p_LCSMngRcp_PLCIdxStat		:= ADR(iPLCIdxStat);
	p_LCSMngRcp_PLCProdRcpInfo	:= ADR(tyPLCProdRcpInfo);
	p_LCSMngRcpProdRcpAct		:= ADR(eProdRcpAct);
	p_LCSMngRcpProdRcpInfoIn	:= ADR(tyProdRcpInfoIn);
	p_LCSMngRcpChkLmt			:= ADR(bChkLmt);

	(* Always Change If Project Change *)

END_PROGRAM
```

#### Act_InitGlobal.st - Change By Project
```iecst
(** 2019-04-24 **)
ACTION Act_InitGlobal:

	(* Always Change If Project Change *)

	//Pass Data To Link
	p_bLinkStartupRun ACCESS p_StartupRun;

	//Pass Data To Internal Use
	p_eAct ACCESS p_LCS_LCSMngRcp_LCSAct;
	p_udiRstErr ACCESS p_RstErrReset;
	p_bPrep ACCESS p_NtParamLCSManageRcpPrep;
	p_bEn ACCESS p_McParamLCSManageRcpEn;
	p_bProdRcpNmExist ACCESS p_ProdRcpNmExist;
	p_bProdRcpNmNotExist ACCESS p_ProdRcpNmNotExist;
	p_bProdRcpNmEmpty ACCESS p_ProdRcpNmEmpty;
	p_bProdRcpListFull ACCESS p_ProdRcpListFull;
	pa_tyProdRcpCurrList ACCESS p_ProdRcpCurrList;
	p_tyProdRcpInfoOut ACCESS p_ProdRcpInfoOut;
	p_tyProdRcpCurrRcp ACCESS p_ProdRcpCurrRcp0;
	p_eProdRcpStat ACCESS p_ProdRcpStat;
	p_eProdRcpStatus ACCESS p_ProdRcpStatus;
	p_sMcParamProdSelRcpNm ACCESS p_ProdRcpCurrRcp0Nm;
	p_diMcParamProdSelWidth ACCESS p_ProdRcpCurrRcp0Width;
	p_iLCSIdxAct ACCESS p_LCS_LCSMngRcp_LCSIdxAct;
	p_iLCSIdxStat ACCESS p_LCS_LCSMngRcp_LCSIdxStat;
	p_tyLCSProdRcpInfo ACCESS p_LCS_LCSMngRcp_LCSProdRcpInfo;
	p_bChkLmtOK ACCESS p_LCSChkLmtOK;
	p_bChkLmtNG ACCESS p_LCSChkLmtNG;
	p_sProgNm ACCESS p_NtParamLCSMngRcpProgNm;
	p_bNtSettingsLoadDone ACCESS p_StartupNtSettingsLoadDone;

	(* Always Change If Project Change *)

END_ACTION
```

#### InputRef_Link.var - Change By Project
```iecst
(*2019-04-24*)
(**)
VAR
	p_bLinkStartupRun : REFERENCE TO BOOL;
END_VAR
```

#### Act_LinkEn.st - Change By Project
```iecst
(** 2019-04-24 **)
ACTION Act_LinkEn:

	//Link bPrep, bEn & bDis
	p_bDis	:= p_bLinkStartupRun;

END_ACTION
```

#### Act_Link.st - Change By Project
```iecst
(** 2019-04-24 **)
ACTION Act_Link:

END_ACTION
```

#### Cyclic.st - Do Not Change!!!
```iecst
(** 2019-04-24 **)
PROGRAM _CYCLIC

	IF bInitDone = FALSE THEN
		bInitDone	:= TRUE;

		Act_InitLocal;
		Act_InitGlobal;

	ELSIF bInitialDone = FALSE THEN
		IF p_bNtSettingsLoadDone = TRUE THEN
			bInitialDone	:= TRUE;

			Act_Initial;
		END_IF

	ELSE

		Act_RstErr;
		Act_LinkAction;
		Act_Action;
		Act_LinkEn;

		IF (p_bPrep = TRUE) AND (p_bEn = TRUE) AND (p_bDis = FALSE) THEN
			Act_Link;
			Act_Background;
			Act_Main;

		ELSE
			Act_Main_Disable;

			IF eStat <> LCSActIdle THEN
				eStatus			:= Done;
				udiPLCStatus	:= 10001;	//LCS Manage Recipe Disabled
			ELSE
				eStatus	:= Idle;
			END_IF
		END_IF

		Act_Alarm;

	END_IF

END_PROGRAM
```

#### Act_InitLocal.st - Do Not Change!!!
```iecst
(** 2019-04-24 **)
ACTION Act_InitLocal:

	//Input Reference Link To Local Variable
	p_eAct ACCESS ADR(eAct);
	p_udiRstErr ACCESS ADR(udiRstErr);
	p_bPrep ACCESS ADR(bPrep);
	p_bEn ACCESS ADR(bEn);
	p_bDis ACCESS ADR(bDis);
	p_bProdRcpNmExist ACCESS ADR(bProdRcpNmExist);
	p_bProdRcpNmNotExist ACCESS ADR(bProdRcpNmNotExist);
	p_bProdRcpNmEmpty ACCESS ADR(bProdRcpNmEmpty);
	p_bProdRcpListFull ACCESS ADR(bProdRcpListFull);
	pa_tyProdRcpCurrList ACCESS ADR(a_tyProdRcpCurrList);
	p_tyProdRcpInfoOut ACCESS ADR(tyProdRcpInfoOut);
	p_tyProdRcpCurrRcp ACCESS ADR(tyProdRcpCurrRcp);
	p_eProdRcpStat ACCESS ADR(eProdRcpStat);
	p_eProdRcpStatus ACCESS ADR(eProdRcpStatus);
	p_sMcParamProdSelRcpNm ACCESS ADR(sMcParamProdSelRcpNm);
	p_diMcParamProdSelWidth ACCESS ADR(diMcParamProdSelWidth);
	p_iLCSIdxAct ACCESS ADR(iLCSIdxAct);
	p_iLCSIdxStat ACCESS ADR(iLCSIdxStat);
	p_tyLCSProdRcpInfo ACCESS ADR(tyLCSProdRcpInfo);
	p_bChkLmtOK ACCESS ADR(bChkLmtOK);
	p_bChkLmtNG ACCESS ADR(bChkLmtNG);
	p_sProgNm ACCESS ADR(sProgNm);
	p_bNtSettingsLoadDone ACCESS ADR(bNtSettingsLoadDone);

END_ACTION
```

#### Act_Initial.st - Do Not Change!!!
```iecst
(** 2019-04-24 **)
ACTION Act_Initial:

	//Initial
	sStatTxt	:= a_sStatText[eStat];

END_ACTION
```

#### Act_Action.st - Do Not Change!!!
```iecst
(** 2019-04-30 **)
ACTION Act_Action:

	//Reset Error
	IF (eStatus = Error) AND bRstErr THEN
		p_eAct	:= LCSActIdle;
		eStat	:= LCSActIdle;
	END_IF

	//Set p_eAct
	IF eStatus = Idle OR eStatus = Busy OR eStatus = Done THEN
		eStat	:= p_eAct;
	END_IF

END_ACTION
```

#### Act_Main.st - Do Not Change!!!
```iecst
(** 2019-04-24 **)
ACTION Act_Main:

	//Main
	CASE eStat OF

		LCSActIdle:
			IF eStatus <> Idle THEN	//Reset Data
				//Private
				eProdRcpAct		:= ProdRcpActIdle;
				usiStep			:= 0;
				iPLCIdxAct		:= 0;
				iPLCIdxStat		:= 0;
				bChkLmt			:= FALSE;

				sStatTxt		:= a_sStatText[eStat];

			END_IF

			eStatus			:= Idle;
			udiPLCStatus	:= 65534;

		LCSActAddProd:
			IF eStatus = Idle OR eStatus = Busy THEN

				eStatus			:= Busy;
				udiPLCStatus	:= 65535;

				sStatTxt	:= a_sStatText[eStat];

				CASE usiStep OF
					0:
						bChkLmt	:= TRUE;

						IF p_bChkLmtOK = TRUE THEN
							usiStep			:= 1;
						ELSIF p_bChkLmtNG = TRUE THEN
							eStatus			:= Done;
							udiPLCStatus	:= 10011;	//Out Of Range While Managing Product
						END_IF

					1:
						tyProdRcpInfoIn	:= p_tyLCSProdRcpInfo;
						eProdRcpAct		:= ProdRcpActAdd;

						IF (p_eProdRcpStat = ProdRcpActAdd) AND (p_eProdRcpStatus = Done) THEN
							eStatus		:= Done;

							IF p_bProdRcpNmEmpty = TRUE THEN
								udiPLCStatus	:= 10012;	//Recipe Name Empty While Adding Product
							ELSIF p_bProdRcpListFull = TRUE THEN
								udiPLCStatus	:= 10013;	//Recipe List Full While Adding Product
							ELSIF p_bProdRcpNmExist = TRUE THEN
								udiPLCStatus	:= 10014;	//Recipe Name Exist While Adding Product
							ELSE
								udiPLCStatus	:= 0;
							END_IF

							eProdRcpAct	:= ProdRcpActIdle;

						ELSIF p_eProdRcpStatus = Error THEN
							eStatus			:= Done;
							udiPLCStatus	:= 10015;	//Recipe Program Error While Adding Product
						END_IF

				END_CASE

			END_IF

		LCSActAddMultiProd:
			IF eStatus = Idle OR eStatus = Busy THEN

				eStatus			:= Busy;
				udiPLCStatus	:= 65535;

				sStatTxt	:= a_sStatText[eStat];

				IF (p_iLCSIdxAct <> 0) THEN
					IF p_iLCSIdxAct <> iPLCIdxStat THEN

						CASE usiStep OF
							0:
								bChkLmt	:= TRUE;

								IF p_bChkLmtOK = TRUE THEN
									usiStep			:= 1;
								ELSIF p_bChkLmtNG = TRUE THEN
									eStatus			:= Done;
									udiPLCStatus	:= 10016;	//Check Limit Error While Adding Multiple Product
								END_IF

							1:
								tyProdRcpInfoIn	:= p_tyLCSProdRcpInfo;
								eProdRcpAct		:= ProdRcpActAdd;

								IF (p_eProdRcpStat = ProdRcpActAdd) AND (p_eProdRcpStatus = Done) THEN
									IF p_bProdRcpNmEmpty = TRUE THEN
										eStatus			:= Done;
										udiPLCStatus	:= 10017;	//Recipe Name Empty While Adding Multiple Product
									ELSIF p_bProdRcpListFull = TRUE THEN
										eStatus			:= Done;
										udiPLCStatus	:= 10018;	//Recipe List Full While Adding Multiple Product
									ELSIF p_bProdRcpNmExist = TRUE THEN
										eStatus			:= Done;
										udiPLCStatus	:= 10019;	//Recipe Name Exist While Adding Multiple Product
									ELSE
										iPLCIdxStat	:= p_iLCSIdxAct;
										usiStep		:= 0;
									END_IF

									eProdRcpAct	:= ProdRcpActIdle;

								ELSIF p_eProdRcpStatus = Error THEN
									eStatus			:= Done;
									udiPLCStatus	:= 10020;	//Recipe Program Error While Adding Multiple Product
								END_IF

						END_CASE

					END_IF

				ELSE
					eStatus			:= Done;
					udiPLCStatus	:= 0;

				END_IF

			END_IF

		LCSActEditProd:
			IF eStatus = Idle OR eStatus = Busy THEN

				eStatus			:= Busy;
				udiPLCStatus	:= 65535;

				sStatTxt	:= a_sStatText[eStat];

				CASE usiStep OF
					0:
						bChkLmt	:= TRUE;

						IF p_bChkLmtOK = TRUE THEN
							usiStep			:= 1;
						ELSIF p_bChkLmtNG = TRUE THEN
							eStatus			:= Done;
							udiPLCStatus	:= 10021;	//Check Limit Error While Editing Product
						END_IF

					1:
						eProdRcpAct	:= ProdRcpActGetInfo;

						IF (p_eProdRcpStat = ProdRcpActGetInfo) AND (p_eProdRcpStatus = Done) THEN

							IF p_tyProdRcpInfoOut.dtLastModified > p_tyLCSProdRcpInfo.dtLastModified THEN
								eStatus			:= Done;
								udiPLCStatus	:= 10049;	//Local Recipe Is Latest Compare With LCS Recipe While Editing Product
							ELSE
								eProdRcpAct	:= ProdRcpActIdle;
								usiStep		:= 2;
							END_IF

						ELSIF p_eProdRcpStatus = Error THEN
							eStatus			:= Done;
							udiPLCStatus	:= 10048;	//Get Recipe Info Error While Editing Product
						END_IF

					2:
						tyProdRcpInfoIn	:= p_tyLCSProdRcpInfo;
						eProdRcpAct		:= ProdRcpActEdit;

						IF (p_eProdRcpStat = ProdRcpActEdit) AND (p_eProdRcpStatus = Done) THEN
							eStatus		:= Done;

							IF p_bProdRcpNmEmpty = TRUE THEN
								udiPLCStatus	:= 10022;	//Recipe Name Empty While Editing Product
							ELSIF p_bProdRcpNmNotExist = TRUE THEN
								udiPLCStatus	:= 10023;	//Recipe Name Not Exist While Editing Product
							ELSE
								udiPLCStatus	:= 0;
							END_IF

							eProdRcpAct	:= ProdRcpActIdle;

						ELSIF p_eProdRcpStatus = Error THEN
							eStatus			:= Done;
							udiPLCStatus	:= 10024;	//Recipe Program Error While Editing Product
						END_IF

				END_CASE

			END_IF

		LCSActEditMultiProd:
			IF eStatus = Idle OR eStatus = Busy THEN

				eStatus			:= Busy;
				udiPLCStatus	:= 65535;

				sStatTxt	:= a_sStatText[eStat];

				IF (p_iLCSIdxAct <> 0) THEN
					IF p_iLCSIdxAct <> iPLCIdxStat THEN

						CASE usiStep OF
							0:
								bChkLmt	:= TRUE;

								IF p_bChkLmtOK = TRUE THEN
									usiStep			:= 1;
								ELSIF p_bChkLmtNG = TRUE THEN
									eStatus			:= Done;
									udiPLCStatus	:= 10025;	//Check Limit Error While Editing Multiple Product
								END_IF

							1:
								eProdRcpAct	:= ProdRcpActGetInfo;

								IF (p_eProdRcpStat = ProdRcpActGetInfo) AND (p_eProdRcpStatus = Done) THEN

									IF p_tyProdRcpInfoOut.dtLastModified > p_tyLCSProdRcpInfo.dtLastModified THEN
										eStatus			:= Done;
										udiPLCStatus	:= 10050;	//Local Recipe Is Latest Compare With LCS Recipe While Editing Multiple Product
									ELSE
										eProdRcpAct	:= ProdRcpActIdle;
										usiStep		:= 2;
									END_IF

								ELSIF p_eProdRcpStatus = Error THEN
									eStatus			:= Done;
									udiPLCStatus	:= 10051;	//Get Recipe Info Error While Editing Multiple Product
								END_IF

							2:
								tyProdRcpInfoIn	:= p_tyLCSProdRcpInfo;
								eProdRcpAct		:= ProdRcpActEdit;

								IF (p_eProdRcpStat = ProdRcpActEdit) AND (p_eProdRcpStatus = Done) THEN
									IF p_bProdRcpNmEmpty = TRUE THEN
										eStatus			:= Done;
										udiPLCStatus	:= 10026;	//Recipe Name Empty While Editing Multiple Product
									ELSIF p_bProdRcpNmNotExist = TRUE THEN
										eStatus			:= Done;
										udiPLCStatus	:= 10027;	//Recipe Name Not Exist While Editing Multiple Product
									ELSE
										iPLCIdxStat	:= p_iLCSIdxAct;
										usiStep		:= 0;
									END_IF

									eProdRcpAct	:= ProdRcpActIdle;

								ELSIF p_eProdRcpStatus = Error THEN
									eStatus			:= Done;
									udiPLCStatus	:= 10028;	//Recipe Program Error While Editing Multiple Product
								END_IF

						END_CASE

					END_IF

				ELSE
					eStatus			:= Done;
					udiPLCStatus	:= 0;

				END_IF

			END_IF

		LCSActOverWriteProd:
			IF eStatus = Idle OR eStatus = Busy THEN

				eStatus			:= Busy;
				udiPLCStatus	:= 65535;

				sStatTxt	:= a_sStatText[eStat];

				CASE usiStep OF
					0:
						bChkLmt	:= TRUE;

						IF p_bChkLmtOK = TRUE THEN
							usiStep			:= 1;
						ELSIF p_bChkLmtNG = TRUE THEN
							eStatus			:= Done;
							udiPLCStatus	:= 10029;	//Check Limit Error While Overwriting Product
						END_IF

					1:
						tyProdRcpInfoIn	:= p_tyLCSProdRcpInfo;
						eProdRcpAct		:= ProdRcpActAddEdit;

						IF (p_eProdRcpStat = ProdRcpActAddEdit) AND (p_eProdRcpStatus = Done) THEN
							eStatus		:= Done;

							IF p_bProdRcpNmEmpty = TRUE THEN
								udiPLCStatus	:= 10030;	//Recipe Name Empty While Overwriting Product
							ELSIF p_bProdRcpListFull = TRUE THEN
								udiPLCStatus	:= 10031;	//Recipe List Full While Overwriting Product
							ELSE
								udiPLCStatus	:= 0;
							END_IF

							eProdRcpAct	:= ProdRcpActIdle;

						ELSIF p_eProdRcpStatus = Error THEN
							eStatus			:= Done;
							udiPLCStatus	:= 10032;	//Recipe Program Error While Overwriting Product
						END_IF

				END_CASE

			END_IF

		LCSActOverWriteMultiProd:
			IF eStatus = Idle OR eStatus = Busy THEN

				eStatus			:= Busy;
				udiPLCStatus	:= 65535;

				sStatTxt	:= a_sStatText[eStat];

				IF (p_iLCSIdxAct <> 0) THEN
					IF p_iLCSIdxAct <> iPLCIdxStat THEN

						CASE usiStep OF
							0:
								bChkLmt	:= TRUE;

								IF p_bChkLmtOK = TRUE THEN
									usiStep			:= 1;
								ELSIF p_bChkLmtNG = TRUE THEN
									eStatus			:= Done;
									udiPLCStatus	:= 10033;	//Check Limit Error While Overwriting Multiple Product
								END_IF

							1:
								tyProdRcpInfoIn	:= p_tyLCSProdRcpInfo;
								eProdRcpAct		:= ProdRcpActAddEdit;

								IF (p_eProdRcpStat = ProdRcpActAddEdit) AND (p_eProdRcpStatus = Done) THEN
									IF p_bProdRcpNmEmpty = TRUE THEN
										eStatus			:= Done;
										udiPLCStatus	:= 10034;	//Recipe Name Empty While Overwriting Multiple Product
									ELSIF p_bProdRcpListFull = TRUE THEN
										eStatus			:= Done;
										udiPLCStatus	:= 10035;	//Recipe List Full While Overwriting Multiple Product
									ELSE
										iPLCIdxStat	:= p_iLCSIdxAct;
										usiStep		:= 0;
									END_IF

									eProdRcpAct	:= ProdRcpActIdle;

								ELSIF p_eProdRcpStatus = Error THEN
									eStatus			:= Done;
									udiPLCStatus	:= 10036;	//Recipe Program Error While Overwriting Multiple Product
								END_IF

						END_CASE

					END_IF

				ELSE
					eStatus			:= Done;
					udiPLCStatus	:= 0;

				END_IF

			END_IF

		LCSActDelProd:
			IF eStatus = Idle OR eStatus = Busy THEN

				eStatus			:= Busy;
				udiPLCStatus	:= 65535;

				sStatTxt	:= a_sStatText[eStat];

				CASE usiStep OF
					0:
						bChkLmt	:= TRUE;

						IF p_bChkLmtOK = TRUE THEN
							usiStep			:= 1;
						ELSIF p_bChkLmtNG = TRUE THEN
							eStatus			:= Done;
							udiPLCStatus	:= 10037;	//Check Limit Error While Deleting Product
						END_IF

					1:
						tyProdRcpInfoIn	:= p_tyLCSProdRcpInfo;
						eProdRcpAct		:= ProdRcpActDel;

						IF (p_eProdRcpStat = ProdRcpActDel) AND (p_eProdRcpStatus = Done) THEN
							eStatus		:= Done;

							IF p_bProdRcpNmEmpty = TRUE THEN
								udiPLCStatus	:= 10038;	//Recipe Name Empty While Deleting Product
							ELSIF p_bProdRcpNmNotExist = TRUE THEN
								udiPLCStatus	:= 10039;	//Recipe Name Not Exist While Deleting Product
							ELSE
								udiPLCStatus	:= 0;
							END_IF

							eProdRcpAct	:= ProdRcpActIdle;

						ELSIF p_eProdRcpStatus = Error THEN
							eStatus			:= Done;
							udiPLCStatus	:= 10040;	//Recipe Program Error While Deleting Product
						END_IF

				END_CASE

			END_IF

		LCSActDelMultiProd:
			IF eStatus = Idle OR eStatus = Busy THEN

				eStatus			:= Busy;
				udiPLCStatus	:= 65535;

				sStatTxt	:= a_sStatText[eStat];

				IF (p_iLCSIdxAct <> 0) THEN
					IF p_iLCSIdxAct <> iPLCIdxStat THEN

						CASE usiStep OF
							0:
								bChkLmt	:= TRUE;

								IF p_bChkLmtOK = TRUE THEN
									usiStep			:= 1;
								ELSIF p_bChkLmtNG = TRUE THEN
									eStatus			:= Done;
									udiPLCStatus	:= 10041;	//Check Limit Error While Deleting Multiple Product
								END_IF

							1:
								tyProdRcpInfoIn	:= p_tyLCSProdRcpInfo;
								eProdRcpAct		:= ProdRcpActDel;

								IF (p_eProdRcpStat = ProdRcpActDel) AND (p_eProdRcpStatus = Done) THEN
									IF p_bProdRcpNmEmpty = TRUE THEN
										eStatus			:= Done;
										udiPLCStatus	:= 10042;	//Recipe Name Empty While Deleting Multiple Product
									ELSIF p_bProdRcpNmNotExist = TRUE THEN
										eStatus			:= Done;
										udiPLCStatus	:= 10043;	//Recipe Name Not Exist While Deleting Multiple Product
									ELSE
										iPLCIdxStat	:= p_iLCSIdxAct;
										usiStep		:= 0;
									END_IF

									eProdRcpAct	:= ProdRcpActIdle;

								ELSIF p_eProdRcpStatus = Error THEN
									eStatus			:= Done;
									udiPLCStatus	:= 10044;	//Recipe Program Error While Deleting Multiple Product
								END_IF

						END_CASE

					END_IF

				ELSE
					eStatus			:= Done;
					udiPLCStatus	:= 0;

				END_IF

			END_IF

		LCSActUploadProd:
			IF eStatus = Idle OR eStatus = Busy THEN

				eStatus			:= Busy;
				udiPLCStatus	:= 65535;

				sStatTxt	:= a_sStatText[eStat];

				tyProdRcpInfoIn	:= p_tyLCSProdRcpInfo;
				eProdRcpAct		:= ProdRcpActGetInfo;

				IF (p_eProdRcpStat = ProdRcpActGetInfo) AND (p_eProdRcpStatus = Done) THEN
					eStatus		:= Done;

					IF p_bProdRcpNmEmpty = TRUE THEN
						udiPLCStatus	:= 10045;	//Recipe Name Empty While Uploading Product
					ELSIF p_bProdRcpNmNotExist = TRUE THEN
						eStatus			:= Done;
						udiPLCStatus	:= 10046;	//Recipe Name Not Exist While Uploading Product
					ELSE
						udiPLCStatus		:= 0;
						tyPLCProdRcpInfo	:= p_tyProdRcpInfoOut;
					END_IF

					eProdRcpAct	:= ProdRcpActIdle;

				ELSIF p_eProdRcpStatus = Error THEN
					eStatus			:= Done;
					udiPLCStatus	:= 10047;	//Recipe Program Error While Uploading Product
				END_IF

			END_IF

		LCSActUploadMultiProd:
			IF eStatus = Idle OR eStatus = Busy THEN

				eStatus			:= Busy;
				udiPLCStatus	:= 65535;

				sStatTxt	:= a_sStatText[eStat];

				IF (iPLCIdxAct = p_iLCSIdxStat) OR (iPLCIdxAct = 0) THEN

					IF pa_tyProdRcpCurrList[iPLCIdxAct + 1].sRcpNm <> '' THEN

						tyPLCProdRcpInfo	:= pa_tyProdRcpCurrList[iPLCIdxAct + 1];
						iPLCIdxAct			:= iPLCIdxAct + 1;

					ELSE

						eStatus			:= Done;
						udiPLCStatus	:= 0;
						iPLCIdxAct		:= 0;

					END_IF

				END_IF

			END_IF

		ELSE
			IF eStatus = Idle OR eStatus = Busy THEN
				eStatus	:= Done;
			END_IF

	END_CASE

END_ACTION
```

#### Act_Background.st - Do Not Change!!!
```iecst
(** 2019-04-24 **)
ACTION Act_Background:

END_ACTION
```

#### Act_Alarm.st - Do Not Change!!!
```iecst
(** 2019-04-24 **)
ACTION Act_Alarm:

	//Error
	IF EDGEPOS(eStatus = Error) THEN

		tyAlmData.sProgNm		:= p_sProgNm;
		tyAlmData.udiCode		:= udiStatus;
		tyAlmData.eSeverity		:= AlmSeverityError;
		tyAlmData.udiRunTime	:= tyAlmData.udiRunTime + 1;
		tyAlmData.bAlm			:= TRUE;
		tyAlmData.udiModuleNum  := udiModuleNum;
		g_sLCSMngRcpProgNm		:= p_sProgNm;
		//Get Error Message
		IF tyAlmData.udiCode < 10000 OR tyAlmData.udiCode > 10099 THEN
			tyAlmData.sAlmMsg	:= 'Unknown';
			tyAlmData.sRcyMsg	:= 'Unknown';
		ELSE
			tyAlmData.sAlmMsg	:= a_tyAlmText[tyAlmData.udiCode].sAlmText;
			tyAlmData.sRcyMsg	:= a_tyAlmText[tyAlmData.udiCode].sRcyText;
		END_IF

		sStatTxt	:= tyAlmData.sAlmMsg;

	ELSIF bRstErr AND (tyAlmData.udiCode <> 0) THEN

		tyAlmData.udiCode	:= 0;
		tyAlmData.eSeverity	:= AlmSeverityNA;
		tyAlmData.sAlmMsg	:= '';
		tyAlmData.sRcyMsg	:= '';
		tyAlmData.bAlm			:= FALSE;
		sStatTxt	:= a_sStatText[eStat];

	END_IF

END_ACTION
```

#### InputRef.var - Do Not Change!!!
```iecst
(*2019-04-24*)
(**)
(*General*)
VAR
	p_eAct : REFERENCE TO eLCSAction;
	p_udiRstErr : REFERENCE TO UDINT;
	p_bPrep : REFERENCE TO BOOL;
	p_bEn : REFERENCE TO BOOL;
	p_bDis : REFERENCE TO BOOL;
END_VAR
(**)
(*Configuration*)
VAR
	p_bProdRcpNmExist : REFERENCE TO BOOL;
	p_bProdRcpNmNotExist : REFERENCE TO BOOL;
	p_bProdRcpNmEmpty : REFERENCE TO BOOL;
	p_bProdRcpListFull : REFERENCE TO BOOL;
	pa_tyProdRcpCurrList : REFERENCE TO ARRAY[1..c_udiProdRcpMax] OF tyProdRcpParam;
	p_tyProdRcpInfoOut : REFERENCE TO tyProdRcpParam;
	p_tyProdRcpCurrRcp : REFERENCE TO tyProdRcpParam;
	p_eProdRcpStat : REFERENCE TO eProdRcpAction;
	p_eProdRcpStatus : REFERENCE TO eFBStatus;
	p_sMcParamProdSelRcpNm : REFERENCE TO STRING[15];
	p_diMcParamProdSelWidth : REFERENCE TO DINT;
	p_iLCSIdxAct : REFERENCE TO INT;
	p_iLCSIdxStat : REFERENCE TO INT;
	p_tyLCSProdRcpInfo : REFERENCE TO tyProdRcpParam;
	p_bChkLmtOK : REFERENCE TO BOOL;
	p_bChkLmtNG : REFERENCE TO BOOL;
	p_sProgNm : REFERENCE TO STRING[15];
	p_bNtSettingsLoadDone : REFERENCE TO BOOL;
END_VAR
```

#### Local.var - Do Not Change!!!
```iecst
(*2019-04-30*)
(**)
(*Local Action, State & Status*)
VAR
	eAct : eLCSAction := LCSActIdle;
	eStat : eLCSAction := LCSActIdle;
	eStatus : eFBStatus := Idle;
	udiStatus : UDINT := 0;
	sStatTxt : STRING[200] := '';
	a_sStatText : ARRAY[0..50] OF STRING[200] := ['Idling','Adding Product','Adding Multiple Products','Editing Product','Editing Multiple Products','OverWrite Product','OverWrite Multiple Products','Deleting Product','Deleting Multiple Products','Running LCS Product','Uploading Product','Uploading Multiple Products',39('')];
END_VAR
(**)
(*Local Alarm*)
VAR
	tyAlmData : tyAlmDat;
	a_tyAlmText : ARRAY[10000..10099] OF tyAlmTxt;
END_VAR
(**)
(*Local Output*)
VAR
	udiPLCStatus : UDINT;
	iPLCIdxAct : INT;
	iPLCIdxStat : INT;
	tyPLCProdRcpInfo : tyProdRcpParam;
	eProdRcpAct : eProdRcpAction;
	tyProdRcpInfoIn : tyProdRcpParam;
	bChkLmt : BOOL;
END_VAR
(**)
(*Local Input*)
VAR
	udiRstErr : UDINT := 0;
	bPrep : BOOL := TRUE;
	bEn : BOOL := TRUE;
	bDis : BOOL := FALSE;
	bProdRcpNmExist : BOOL;
	bProdRcpNmNotExist : BOOL;
	bProdRcpNmEmpty : BOOL;
	bProdRcpListFull : BOOL;
	a_tyProdRcpCurrList : ARRAY[1..c_udiProdRcpMax] OF tyProdRcpParam;
	tyProdRcpInfoOut : tyProdRcpParam;
	tyProdRcpCurrRcp : tyProdRcpParam;
	eProdRcpStat : eProdRcpAction;
	eProdRcpStatus : eFBStatus;
	sMcParamProdSelRcpNm : STRING[15];
	diMcParamProdSelWidth : DINT;
	iLCSIdxAct : INT;
	iLCSIdxStat : INT;
	tyLCSProdRcpInfo : tyProdRcpParam;
	bChkLmtOK : BOOL;
	bChkLmtNG : BOOL;
	sProgNm : STRING[15] := 'LCSMngRcp';
	bNtSettingsLoadDone : BOOL := TRUE;
END_VAR
(**)
(*Local*)
VAR
	bRstErr : BOOL;
	udiRstErrOld : UDINT;
	bInitDone : BOOL;
	bInitialDone : BOOL;
	usiStep : USINT;
	udiModuleNum : UDINT := 4201;
END_VAR
```

### LCSLF.var - Change By Project
```iecst
(*2019-06-12*)
(**)
(*Action & State & Status*)
VAR
	p_LCSLFStat : UDINT;
	p_LCSLFStatus : UDINT;
	p_LCSLFStatTxt : UDINT;
END_VAR
(**)
(*Alarm*)
VAR
	p_LCSLFAlmData : UDINT;
	p_LCSLFInfoData : UDINT;
END_VAR
(**)
(*Output*)
VAR
	p_LCSLF_PLCStatus : UDINT;
	p_LCSLFChkLmt : UDINT;
	p_LCSLFAccDataMnl : UDINT;
	p_LCSLFUpdtDataMnl : UDINT;
	p_LCSLFUpdtProdRcpNm : UDINT;
	p_LCSLFUpdtProdWidth : UDINT;
END_VAR
```
